LIN {X 0,Y 573.635,Z 572.354,A -85,B 0,C 180,E1 -2236.63,E2 -2236.63} C_VEL
LIN {X 0,Y 573.477,Z 582.752,A -85,B 0,C 180,E1 -2237.616,E2 -2237.616} C_VEL
LIN {X 0,Y 573.285,Z 592.771,A -85,B 0,C 180,E1 -2238.734,E2 -2238.734} C_VEL
LIN {X 0,Y 573.242,Z 601.859,A -85,B 0,C 180,E1 -2239.939,E2 -2239.939} C_VEL
LIN {X 0,Y 573.133,Z 609.735,A -85,B 0,C 180,E1 -2241.183,E2 -2241.183} C_VEL
LIN {X 0,Y 573.074,Z 617.09,A -85,B 0,C 180,E1 -2242.602,E2 -2242.602} C_VEL
LIN {X 0,Y 573.04,Z 622.924,A -85,B 0,C 180,E1 -2244.016,E2 -2244.016} C_VEL
LIN {X 0,Y 572.951,Z 626.386,A -85,B 0,C 180,E1 -2245.074,E2 -2245.074} C_VEL
LIN {X 0,Y 573.004,Z 629.889,A -85,B 0,C 180,E1 -2246.484,E2 -2246.484} C_VEL
LIN {X 0,Y 572.937,Z 632.192,A -85,B 0,C 180,E1 -2247.891,E2 -2247.891} C_VEL
LIN {X 0,Y 572.938,Z 633.349,A -85,B 0,C 180,E1 -2249.297,E2 -2249.297} C_VEL
LIN {X 0,Y 572.938,Z 633.349,A -85,B 0,C 180,E1 -2250.703,E2 -2250.703} C_VEL
LIN {X 0,Y 572.937,Z 632.191,A -85,B 0,C 180,E1 -2252.109,E2 -2252.109} C_VEL
LIN {X 0,Y 573.004,Z 629.887,A -85,B 0,C 180,E1 -2253.516,E2 -2253.516} C_VEL
LIN {X 0,Y 572.951,Z 626.386,A -85,B 0,C 180,E1 -2254.926,E2 -2254.926} C_VEL
LIN {X 0,Y 573.012,Z 621.609,A -85,B 0,C 180,E1 -2256.337,E2 -2256.337} C_VEL
LIN {X 0,Y 573.093,Z 615.424,A -85,B 0,C 180,E1 -2257.752,E2 -2257.752} C_VEL
LIN {X 0,Y 573.136,Z 607.65,A -85,B 0,C 180,E1 -2259.172,E2 -2259.172} C_VEL
LIN {X 0,Y 573.27,Z 599.371,A -85,B 0,C 180,E1 -2260.418,E2 -2260.418} C_VEL
LIN {X 0,Y 573.385,Z 589.394,A -85,B 0,C 180,E1 -2261.668,E2 -2261.668} C_VEL
LIN {X 0,Y 573.568,Z 579.192,A -85,B 0,C 180,E1 -2262.741,E2 -2262.741} C_VEL
LIN {X 0,Y 573.742,Z 567.024,A -85,B 0,C 180,E1 -2263.819,E2 -2263.819} C_VEL
LIN {X 0,Y 573.961,Z 553.91,A -85,B 0,C 180,E1 -2264.781,E2 -2264.781} C_VEL
LIN {X 0,Y 574.143,Z 539.88,A -85,B 0,C 180,E1 -2265.622,E2 -2265.622} C_VEL
LIN {X 0,Y 574.334,Z 525.81,A -85,B 0,C 180,E1 -2266.3,E2 -2266.3} C_VEL
LIN {X 0,Y 574.562,Z 511.319,A -85,B 0,C 180,E1 -2266.842,E2 -2266.842} C_VEL
LIN {X 0,Y 574.705,Z 496.022,A -85,B 0,C 180,E1 -2267.261,E2 -2267.261} C_VEL
LIN {X 0,Y 574.796,Z 480.66,A -85,B 0,C 180,E1 -2267.532,E2 -2267.532} C_VEL
LIN {X 0,Y 575.14,Z 327.837,A -85,B 0,C 180,E1 -2269.493,E2 -2269.493} C_VEL
LIN {X 0,Y 574.002,Z 321.813,A -85,B 0,C 180,E1 -2269.623,E2 -2269.623} C_VEL
LIN {X 0,Y 574.348,Z 296.397,A -85,B 0,C 180,E1 -2272.671,E2 -2272.671} C_VEL
LIN {X 0,Y 574.606,Z 274.457,A -85,B 0,C 180,E1 -2275.345,E2 -2275.345} C_VEL
LIN {X 0,Y 574.309,Z 271.29,A -85,B 0,C 180,E1 -2275.748,E2 -2275.748} C_VEL
LIN {X 0,Y 573.237,Z 266.71,A -85,B 0,C 180,E1 -2276.376,E2 -2276.376} C_VEL
LIN {X 0,Y 573.255,Z 266.699,A -85,B 0,C 180,E1 -2279.365,E2 -2279.365} C_VEL
LIN {X 0,Y 573.242,Z 266.707,A -85,B 0,C 180,E1 -2282.227,E2 -2282.227} C_VEL
LIN {X 0,Y 573.219,Z 266.703,A -85,B 0,C 180,E1 -2284.769,E2 -2284.769} C_VEL
LIN {X 0,Y 573.216,Z 266.708,A -85,B 0,C 180,E1 -2287.808,E2 -2287.808} C_VEL
LIN {X 0,Y 573.238,Z 266.703,A -85,B 0,C 180,E1 -2290.524,E2 -2290.524} C_VEL
LIN {X 0,Y 573.19,Z 266.707,A -85,B 0,C 180,E1 -2293.362,E2 -2293.362} C_VEL
LIN {X 0,Y 573.2,Z 266.709,A -85,B 0,C 180,E1 -2296.334,E2 -2296.334} C_VEL
LIN {X 0,Y 573.198,Z 266.706,A -85,B 0,C 180,E1 -2298.54,E2 -2298.54} C_VEL
LIN {X 0,Y 573.221,Z 266.703,A -85,B 0,C 180,E1 -2301.297,E2 -2301.297} C_VEL
LIN {X 0,Y 573.173,Z 266.715,A -85,B 0,C 180,E1 -2304.022,E2 -2304.022} C_VEL
LIN {X 0,Y 573.218,Z 266.702,A -85,B 0,C 180,E1 -2306.514,E2 -2306.514} C_VEL
LIN {X 0,Y 573.208,Z 266.704,A -85,B 0,C 180,E1 -2309.119,E2 -2309.119} C_VEL
LIN {X 0,Y 573.207,Z 266.709,A -85,B 0,C 180,E1 -2311.977,E2 -2311.977} C_VEL
LIN {X 0,Y 573.192,Z 266.705,A -85,B 0,C 180,E1 -2314.587,E2 -2314.587} C_VEL
LIN {X 0,Y 573.222,Z 266.702,A -85,B 0,C 180,E1 -2316.9,E2 -2316.9} C_VEL
LIN {X 0,Y 573.233,Z 266.703,A -85,B 0,C 180,E1 -2319.173,E2 -2319.173} C_VEL
LIN {X 0,Y 573.186,Z 266.709,A -85,B 0,C 180,E1 -2321.41,E2 -2321.41} C_VEL
LIN {X 0,Y 573.2,Z 266.705,A -85,B 0,C 180,E1 -2324.351,E2 -2324.351} C_VEL
LIN {X 0,Y 573.187,Z 266.705,A -85,B 0,C 180,E1 -2326.528,E2 -2326.528} C_VEL
LIN {X 0,Y 573.212,Z 266.706,A -85,B 0,C 180,E1 -2329.402,E2 -2329.402} C_VEL
LIN {X 0,Y 573.196,Z 266.705,A -85,B 0,C 180,E1 -2332.249,E2 -2332.249} C_VEL
LIN {X 0,Y 573.246,Z 266.697,A -85,B 0,C 180,E1 -2334.371,E2 -2334.371} C_VEL
LIN {X 0,Y 573.283,Z 266.7,A -85,B 0,C 180,E1 -2337.189,E2 -2337.189} C_VEL
LIN {X 0,Y 573.285,Z 266.695,A -85,B 0,C 180,E1 -2340,E2 -2340} C_VEL
LIN {X 0,Y 573.272,Z 266.697,A -85,B 0,C 180,E1 -2342.811,E2 -2342.811} C_VEL
LIN {X 0,Y 573.27,Z 266.7,A -85,B 0,C 180,E1 -2345.628,E2 -2345.628} C_VEL
LIN {X 0,Y 573.251,Z 266.701,A -85,B 0,C 180,E1 -2347.751,E2 -2347.751} C_VEL
LIN {X 0,Y 573.226,Z 266.702,A -85,B 0,C 180,E1 -2350.597,E2 -2350.597} C_VEL
LIN {X 0,Y 573.21,Z 266.706,A -85,B 0,C 180,E1 -2352.75,E2 -2352.75} C_VEL
LIN {X 0,Y 573.207,Z 266.709,A -85,B 0,C 180,E1 -2354.921,E2 -2354.921} C_VEL
LIN {X 0,Y 573.22,Z 266.702,A -85,B 0,C 180,E1 -2357.849,E2 -2357.849} C_VEL
LIN {X 0,Y 573.221,Z 266.698,A -85,B 0,C 180,E1 -2360.078,E2 -2360.078} C_VEL
LIN {X 0,Y 573.208,Z 266.702,A -85,B 0,C 180,E1 -2362.339,E2 -2362.339} C_VEL
LIN {X 0,Y 573.2,Z 266.705,A -85,B 0,C 180,E1 -2364.352,E2 -2364.352} C_VEL
LIN {X 0,Y 572.567,Z 266.791,A -85,B 0,C 180,E1 -2364.938,E2 -2364.938} C_VEL
LIN {X 0,Y 569.747,Z 267.143,A -85,B 0,C 180,E1 -2365.89,E2 -2365.89} C_VEL
LIN {X 0,Y 567.336,Z 267.442,A -85,B 0,C 180,E1 -2366.656,E2 -2366.656} C_VEL
LIN {X 0,Y 566.283,Z 267.569,A -85,B 0,C 180,E1 -2367.247,E2 -2367.247} C_VEL
LIN {X 0,Y 566.19,Z 267.578,A -85,B 0,C 180,E1 -2367.447,E2 -2367.447} C_VEL
LIN {X 0,Y 566.185,Z 267.578,A -85,B 0,C 180,E1 -2369.77,E2 -2369.77} C_VEL
LIN {X 0,Y 566.191,Z 267.579,A -85,B 0,C 180,E1 -2372.43,E2 -2372.43} C_VEL
LIN {X 0,Y 566.173,Z 267.588,A -85,B 0,C 180,E1 -2374.991,E2 -2374.991} C_VEL
LIN {X 0,Y 566.186,Z 267.579,A -85,B 0,C 180,E1 -2377.462,E2 -2377.462} C_VEL
LIN {X 0,Y 566.198,Z 267.577,A -85,B 0,C 180,E1 -2380.2,E2 -2380.2} C_VEL
LIN {X 0,Y 566.193,Z 267.583,A -85,B 0,C 180,E1 -2383.055,E2 -2383.055} C_VEL
LIN {X 0,Y 566.187,Z 267.579,A -85,B 0,C 180,E1 -2386.05,E2 -2386.05} C_VEL
LIN {X 0,Y 566.197,Z 267.58,A -85,B 0,C 180,E1 -2389.216,E2 -2389.216} C_VEL
LIN {X 0,Y 566.176,Z 267.579,A -85,B 0,C 180,E1 -2391.637,E2 -2391.637} C_VEL
LIN {X 0,Y 566.169,Z 267.585,A -85,B 0,C 180,E1 -2394.31,E2 -2394.31} C_VEL
LIN {X 0,Y 566.2,Z 267.583,A -85,B 0,C 180,E1 -2396.898,E2 -2396.898} C_VEL
LIN {X 0,Y 566.175,Z 267.581,A -85,B 0,C 180,E1 -2399.408,E2 -2399.408} C_VEL
LIN {X 0,Y 566.21,Z 267.577,A -85,B 0,C 180,E1 -2401.858,E2 -2401.858} C_VEL
LIN {X 0,Y 566.209,Z 267.582,A -85,B 0,C 180,E1 -2404.252,E2 -2404.252} C_VEL
LIN {X 0,Y 566.227,Z 267.735,A -85,B 0,C 180,E1 -2406.574,E2 -2406.574} C_VEL
LIN {X 0,Y 567.168,Z 273.21,A -85,B 0,C 180,E1 -2407.411,E2 -2407.411} C_VEL
LIN {X 0,Y 566.915,Z 292.519,A -85,B 0,C 180,E1 -2410.134,E2 -2410.134} C_VEL
LIN {X 0,Y 566.916,Z 292.904,A -85,B 0,C 180,E1 -2410.188,E2 -2410.188} C_VEL
LIN {X 0,Y 568.47,Z 301.087,A -85,B 0,C 180,E1 -2410.357,E2 -2410.357} C_VEL
LIN {X 0,Y 567.974,Z 458.169,A -85,B 0,C 180,E1 -2412.413,E2 -2412.413} C_VEL
LIN {X 0,Y 567.827,Z 473.784,A -85,B 0,C 180,E1 -2412.767,E2 -2412.767} C_VEL
LIN {X 0,Y 567.607,Z 489.09,A -85,B 0,C 180,E1 -2413.27,E2 -2413.27} C_VEL
LIN {X 0,Y 567.399,Z 503.742,A -85,B 0,C 180,E1 -2413.911,E2 -2413.911} C_VEL
LIN {X 0,Y 567.146,Z 517.054,A -85,B 0,C 180,E1 -2414.641,E2 -2414.641} C_VEL
LIN {X 0,Y 566.917,Z 529.984,A -85,B 0,C 180,E1 -2415.508,E2 -2415.508} C_VEL
LIN {X 0,Y 566.653,Z 542.893,A -85,B 0,C 180,E1 -2416.553,E2 -2416.553} C_VEL
LIN {X 0,Y 566.479,Z 554.088,A -85,B 0,C 180,E1 -2417.643,E2 -2417.643} C_VEL
LIN {X 0,Y 566.263,Z 564.18,A -85,B 0,C 180,E1 -2418.81,E2 -2418.81} C_VEL
LIN {X 0,Y 566.133,Z 574.006,A -85,B 0,C 180,E1 -2420.172,E2 -2420.172} C_VEL
LIN {X 0,Y 566.064,Z 581.496,A -85,B 0,C 180,E1 -2421.432,E2 -2421.432} C_VEL
LIN {X 0,Y 565.975,Z 588.5,A -85,B 0,C 180,E1 -2422.867,E2 -2422.867} C_VEL
LIN {X 0,Y 565.981,Z 594.009,A -85,B 0,C 180,E1 -2424.299,E2 -2424.299} C_VEL
LIN {X 0,Y 565.914,Z 598.178,A -85,B 0,C 180,E1 -2425.727,E2 -2425.727} C_VEL
LIN {X 0,Y 565.872,Z 601.113,A -85,B 0,C 180,E1 -2427.153,E2 -2427.153} C_VEL
LIN {X 0,Y 565.842,Z 602.879,A -85,B 0,C 180,E1 -2428.577,E2 -2428.577} C_VEL
LIN {X 0,Y 565.837,Z 603.496,A -85,B 0,C 180,E1 -2430,E2 -2430} C_VEL
LIN {X 0,Y 565.844,Z 602.941,A -85,B 0,C 180,E1 -2431.423,E2 -2431.423} C_VEL
LIN {X 0,Y 565.874,Z 601.258,A -85,B 0,C 180,E1 -2432.847,E2 -2432.847} C_VEL
LIN {X 0,Y 565.914,Z 598.404,A -85,B 0,C 180,E1 -2434.273,E2 -2434.273} C_VEL
LIN {X 0,Y 565.975,Z 594.318,A -85,B 0,C 180,E1 -2435.701,E2 -2435.701} C_VEL
LIN {X 0,Y 565.975,Z 588.904,A -85,B 0,C 180,E1 -2437.133,E2 -2437.133} C_VEL
LIN {X 0,Y 566.06,Z 582.004,A -85,B 0,C 180,E1 -2438.568,E2 -2438.568} C_VEL
LIN {X 0,Y 566.177,Z 573.396,A -85,B 0,C 180,E1 -2440.008,E2 -2440.008} C_VEL
LIN {X 0,Y 566.25,Z 564.953,A -85,B 0,C 180,E1 -2441.183,E2 -2441.183} C_VEL
LIN {X 0,Y 566.436,Z 554.917,A -85,B 0,C 180,E1 -2442.358,E2 -2442.358} C_VEL
LIN {X 0,Y 566.668,Z 542.874,A -85,B 0,C 180,E1 -2443.538,E2 -2443.538} C_VEL
LIN {X 0,Y 566.877,Z 531.252,A -85,B 0,C 180,E1 -2444.488,E2 -2444.488} C_VEL
LIN {X 0,Y 567.09,Z 518.478,A -85,B 0,C 180,E1 -2445.361,E2 -2445.361} C_VEL
LIN {X 0,Y 567.377,Z 505.469,A -85,B 0,C 180,E1 -2446.09,E2 -2446.09} C_VEL
LIN {X 0,Y 567.555,Z 491.278,A -85,B 0,C 180,E1 -2446.732,E2 -2446.732} C_VEL
LIN {X 0,Y 567.793,Z 476.732,A -85,B 0,C 180,E1 -2447.235,E2 -2447.235} C_VEL
LIN {X 0,Y 567.922,Z 461.44,A -85,B 0,C 180,E1 -2447.613,E2 -2447.613} C_VEL
LIN {X 0,Y 568.073,Z 439.94,A -85,B 0,C 180,E1 -2447.931,E2 -2447.931} C_VEL
LIN {X 0,Y 568.46,Z 300.582,A -85,B 0,C 180,E1 -2449.74,E2 -2449.74} C_VEL
LIN {X 0,Y 566.883,Z 292.906,A -85,B 0,C 180,E1 -2449.903,E2 -2449.903} C_VEL
LIN {X 0,Y 567.205,Z 275.173,A -85,B 0,C 180,E1 -2452.396,E2 -2452.396} C_VEL
LIN {X 0,Y 566.947,Z 271.258,A -85,B 0,C 180,E1 -2452.973,E2 -2452.973} C_VEL
LIN {X 0,Y 566.211,Z 267.584,A -85,B 0,C 180,E1 -2453.548,E2 -2453.548} C_VEL
LIN {X 0,Y 566.213,Z 267.583,A -85,B 0,C 180,E1 -2455.748,E2 -2455.748} C_VEL
LIN {X 0,Y 566.201,Z 267.579,A -85,B 0,C 180,E1 -2458.201,E2 -2458.201} C_VEL
LIN {X 0,Y 566.191,Z 267.582,A -85,B 0,C 180,E1 -2461.076,E2 -2461.076} C_VEL
LIN {X 0,Y 566.209,Z 267.581,A -85,B 0,C 180,E1 -2463.733,E2 -2463.733} C_VEL
LIN {X 0,Y 566.204,Z 267.577,A -85,B 0,C 180,E1 -2466.568,E2 -2466.568} C_VEL
LIN {X 0,Y 566.215,Z 267.578,A -85,B 0,C 180,E1 -2469.686,E2 -2469.686} C_VEL
LIN {X 0,Y 566.195,Z 267.581,A -85,B 0,C 180,E1 -2472.916,E2 -2472.916} C_VEL
LIN {X 0,Y 566.186,Z 267.579,A -85,B 0,C 180,E1 -2476.048,E2 -2476.048} C_VEL
LIN {X 0,Y 566.195,Z 267.584,A -85,B 0,C 180,E1 -2479.214,E2 -2479.214} C_VEL
LIN {X 0,Y 566.173,Z 267.582,A -85,B 0,C 180,E1 -2481.636,E2 -2481.636} C_VEL
LIN {X 0,Y 566.155,Z 267.58,A -85,B 0,C 180,E1 -2484.307,E2 -2484.307} C_VEL
LIN {X 0,Y 566.193,Z 267.583,A -85,B 0,C 180,E1 -2486.896,E2 -2486.896} C_VEL
LIN {X 0,Y 566.167,Z 267.582,A -85,B 0,C 180,E1 -2489.406,E2 -2489.406} C_VEL
LIN {X 0,Y 566.201,Z 267.576,A -85,B 0,C 180,E1 -2491.857,E2 -2491.857} C_VEL
LIN {X 0,Y 566.193,Z 267.577,A -85,B 0,C 180,E1 -2494.25,E2 -2494.25} C_VEL
LIN {X 0,Y 566.159,Z 267.584,A -85,B 0,C 180,E1 -2497.367,E2 -2497.367} C_VEL
LIN {X 0,Y 566.191,Z 267.578,A -85,B 0,C 180,E1 -2499.662,E2 -2499.662} C_VEL
LIN {X 0,Y 566.183,Z 267.583,A -85,B 0,C 180,E1 -2502.668,E2 -2502.668} C_VEL
LIN {X 0,Y 566.2,Z 267.576,A -85,B 0,C 180,E1 -2505.626,E2 -2505.626} C_VEL
LIN {X 0,Y 566.219,Z 267.581,A -85,B 0,C 180,E1 -2508.676,E2 -2508.676} C_VEL
LIN {X 0,Y 566.178,Z 267.579,A -85,B 0,C 180,E1 -2511.433,E2 -2511.433} C_VEL
LIN {X 0,Y 566.237,Z 267.575,A -85,B 0,C 180,E1 -2514.301,E2 -2514.301} C_VEL
LIN {X 0,Y 566.248,Z 267.571,A -85,B 0,C 180,E1 -2517.866,E2 -2517.866} C_VEL
LIN {X 0,Y 566.291,Z 267.574,A -85,B 0,C 180,E1 -2520.711,E2 -2520.711} C_VEL
LIN {X 0,Y 566.25,Z 267.576,A -85,B 0,C 180,E1 -2522.846,E2 -2522.846} C_VEL
LIN {X 0,Y 566.217,Z 267.574,A -85,B 0,C 180,E1 -2525.699,E2 -2525.699} C_VEL
LIN {X 0,Y 566.168,Z 267.581,A -85,B 0,C 180,E1 -2527.848,E2 -2527.848} C_VEL
LIN {X 0,Y 566.205,Z 267.582,A -85,B 0,C 180,E1 -2530.73,E2 -2530.73} C_VEL
LIN {X 0,Y 566.163,Z 267.58,A -85,B 0,C 180,E1 -2533.642,E2 -2533.642} C_VEL
LIN {X 0,Y 566.168,Z 267.582,A -85,B 0,C 180,E1 -2535.848,E2 -2535.848} C_VEL
LIN {X 0,Y 566.173,Z 267.583,A -85,B 0,C 180,E1 -2538.829,E2 -2538.829} C_VEL
LIN {X 0,Y 566.194,Z 267.577,A -85,B 0,C 180,E1 -2541.42,E2 -2541.42} C_VEL
LIN {X 0,Y 566.155,Z 267.59,A -85,B 0,C 180,E1 -2544.183,E2 -2544.183} C_VEL
LIN {X 0,Y 566.155,Z 267.586,A -85,B 0,C 180,E1 -2546.652,E2 -2546.652} C_VEL
LIN {X 0,Y 566.157,Z 267.583,A -85,B 0,C 180,E1 -2548.955,E2 -2548.955} C_VEL
LIN {X 0,Y 566.176,Z 267.58,A -85,B 0,C 180,E1 -2551.423,E2 -2551.423} C_VEL
LIN {X 0,Y 566.181,Z 267.584,A -85,B 0,C 180,E1 -2553.958,E2 -2553.958} C_VEL
LIN {X 0,Y 566.133,Z 267.588,A -85,B 0,C 180,E1 -2556.575,E2 -2556.575} C_VEL
LIN {X 0,Y 566.195,Z 267.576,A -85,B 0,C 180,E1 -2559.275,E2 -2559.275} C_VEL
LIN {X 0,Y 566.172,Z 267.588,A -85,B 0,C 180,E1 -2562.091,E2 -2562.091} C_VEL
LIN {X 0,Y 566.154,Z 267.582,A -85,B 0,C 180,E1 -2565.038,E2 -2565.038} C_VEL
LIN {X 0,Y 566.161,Z 267.59,A -85,B 0,C 180,E1 -2567.909,E2 -2567.909} C_VEL
LIN {X 0,Y 566.202,Z 267.577,A -85,B 0,C 180,E1 -2570.727,E2 -2570.727} C_VEL
LIN {X 0,Y 566.171,Z 267.583,A -85,B 0,C 180,E1 -2573.429,E2 -2573.429} C_VEL
LIN {X 0,Y 566.206,Z 267.58,A -85,B 0,C 180,E1 -2576.267,E2 -2576.267} C_VEL
LIN {X 0,Y 566.183,Z 267.579,A -85,B 0,C 180,E1 -2578.925,E2 -2578.925} C_VEL
LIN {X 0,Y 566.183,Z 267.588,A -85,B 0,C 180,E1 -2581.857,E2 -2581.857} C_VEL
LIN {X 0,Y 566.163,Z 267.651,A -85,B 0,C 180,E1 -2583.424,E2 -2583.424} C_VEL
LIN {X 0,Y 567.691,Z 274.277,A -85,B 0,C 180,E1 -2584.324,E2 -2584.324} C_VEL
LIN {X 0,Y 567.568,Z 291.067,A -85,B 0,C 180,E1 -2586.393,E2 -2586.393} C_VEL
LIN {X 0,Y 567.282,Z 312.003,A -85,B 0,C 180,E1 -2588.945,E2 -2588.945} C_VEL
LIN {X 0,Y 567.116,Z 321.949,A -85,B 0,C 180,E1 -2590.143,E2 -2590.143} C_VEL
LIN {X 0,Y 568.507,Z 330.374,A -85,B 0,C 180,E1 -2590.304,E2 -2590.304} C_VEL
LIN {X 0,Y 567.994,Z 488.201,A -85,B 0,C 180,E1 -2592.369,E2 -2592.369} C_VEL
LIN {X 0,Y 567.834,Z 503.721,A -85,B 0,C 180,E1 -2592.72,E2 -2592.72} C_VEL
LIN {X 0,Y 567.61,Z 519.05,A -85,B 0,C 180,E1 -2593.223,E2 -2593.223} C_VEL
LIN {X 0,Y 567.444,Z 532.784,A -85,B 0,C 180,E1 -2593.82,E2 -2593.82} C_VEL
LIN {X 0,Y 567.151,Z 546.255,A -85,B 0,C 180,E1 -2594.549,E2 -2594.549} C_VEL
LIN {X 0,Y 566.931,Z 558.527,A -85,B 0,C 180,E1 -2595.359,E2 -2595.359} C_VEL
LIN {X 0,Y 566.671,Z 571.296,A -85,B 0,C 180,E1 -2596.371,E2 -2596.371} C_VEL
LIN {X 0,Y 566.491,Z 582.753,A -85,B 0,C 180,E1 -2597.461,E2 -2597.461} C_VEL
LIN {X 0,Y 566.268,Z 593.314,A -85,B 0,C 180,E1 -2598.659,E2 -2598.659} C_VEL
LIN {X 0,Y 566.208,Z 601.858,A -85,B 0,C 180,E1 -2599.812,E2 -2599.812} C_VEL
LIN {X 0,Y 566.057,Z 609.736,A -85,B 0,C 180,E1 -2601.072,E2 -2601.072} C_VEL
LIN {X 0,Y 565.997,Z 617.091,A -85,B 0,C 180,E1 -2602.509,E2 -2602.509} C_VEL
LIN {X 0,Y 565.956,Z 622.923,A -85,B 0,C 180,E1 -2603.941,E2 -2603.941} C_VEL
LIN {X 0,Y 565.866,Z 626.386,A -85,B 0,C 180,E1 -2605.013,E2 -2605.013} C_VEL
LIN {X 0,Y 565.909,Z 629.89,A -85,B 0,C 180,E1 -2606.44,E2 -2606.44} C_VEL
LIN {X 0,Y 565.838,Z 632.192,A -85,B 0,C 180,E1 -2607.865,E2 -2607.865} C_VEL
LIN {X 0,Y 565.838,Z 633.349,A -85,B 0,C 180,E1 -2609.288,E2 -2609.288} C_VEL
LIN {X 0,Y 565.838,Z 633.348,A -85,B 0,C 180,E1 -2610.712,E2 -2610.712} C_VEL
LIN {X 0,Y 565.838,Z 632.19,A -85,B 0,C 180,E1 -2612.135,E2 -2612.135} C_VEL
LIN {X 0,Y 565.909,Z 629.887,A -85,B 0,C 180,E1 -2613.56,E2 -2613.56} C_VEL
LIN {X 0,Y 565.866,Z 626.386,A -85,B 0,C 180,E1 -2614.987,E2 -2614.987} C_VEL
LIN {X 0,Y 565.956,Z 622.925,A -85,B 0,C 180,E1 -2616.059,E2 -2616.059} C_VEL
LIN {X 0,Y 565.997,Z 617.089,A -85,B 0,C 180,E1 -2617.491,E2 -2617.491} C_VEL
LIN {X 0,Y 566.057,Z 609.732,A -85,B 0,C 180,E1 -2618.928,E2 -2618.928} C_VEL
LIN {X 0,Y 566.208,Z 601.858,A -85,B 0,C 180,E1 -2620.188,E2 -2620.188} C_VEL
LIN {X 0,Y 566.308,Z 592.393,A -85,B 0,C 180,E1 -2621.453,E2 -2621.453} C_VEL
LIN {X 0,Y 566.491,Z 582.752,A -85,B 0,C 180,E1 -2622.539,E2 -2622.539} C_VEL
LIN {X 0,Y 566.672,Z 571.299,A -85,B 0,C 180,E1 -2623.629,E2 -2623.629} C_VEL
LIN {X 0,Y 566.948,Z 558.683,A -85,B 0,C 180,E1 -2624.63,E2 -2624.63} C_VEL
LIN {X 0,Y 567.151,Z 546.253,A -85,B 0,C 180,E1 -2625.451,E2 -2625.451} C_VEL
LIN {X 0,Y 567.461,Z 532.778,A -85,B 0,C 180,E1 -2626.18,E2 -2626.18} C_VEL
LIN {X 0,Y 567.639,Z 519.058,A -85,B 0,C 180,E1 -2626.776,E2 -2626.776} C_VEL
LIN {X 0,Y 567.847,Z 503.735,A -85,B 0,C 180,E1 -2627.279,E2 -2627.279} C_VEL
LIN {X 0,Y 567.98,Z 488.315,A -85,B 0,C 180,E1 -2627.63,E2 -2627.63} C_VEL
LIN {X 0,Y 568.493,Z 329.51,A -85,B 0,C 180,E1 -2629.708,E2 -2629.708} C_VEL
LIN {X 0,Y 567.135,Z 321.838,A -85,B 0,C 180,E1 -2629.867,E2 -2629.867} C_VEL
LIN {X 0,Y 567.548,Z 294.798,A -85,B 0,C 180,E1 -2633.151,E2 -2633.151} C_VEL
LIN {X 0,Y 567.795,Z 276.046,A -85,B 0,C 180,E1 -2635.452,E2 -2635.452} C_VEL
LIN {X 0,Y 567.025,Z 271.103,A -85,B 0,C 180,E1 -2636.103,E2 -2636.103} C_VEL
LIN {X 0,Y 566.15,Z 267.591,A -85,B 0,C 180,E1 -2636.598,E2 -2636.598} C_VEL
LIN {X 0,Y 566.178,Z 267.581,A -85,B 0,C 180,E1 -2638.953,E2 -2638.953} C_VEL
LIN {X 0,Y 566.185,Z 267.579,A -85,B 0,C 180,E1 -2641.421,E2 -2641.421} C_VEL
LIN {X 0,Y 566.202,Z 267.584,A -85,B 0,C 180,E1 -2643.955,E2 -2643.955} C_VEL
LIN {X 0,Y 566.171,Z 267.583,A -85,B 0,C 180,E1 -2646.571,E2 -2646.571} C_VEL
LIN {X 0,Y 566.204,Z 267.581,A -85,B 0,C 180,E1 -2649.684,E2 -2649.684} C_VEL
LIN {X 0,Y 566.174,Z 267.58,A -85,B 0,C 180,E1 -2652.914,E2 -2652.914} C_VEL
LIN {X 0,Y 566.15,Z 267.592,A -85,B 0,C 180,E1 -2656.052,E2 -2656.052} C_VEL
LIN {X 0,Y 566.149,Z 267.583,A -85,B 0,C 180,E1 -2658.858,E2 -2658.858} C_VEL
LIN {X 0,Y 566.191,Z 267.581,A -85,B 0,C 180,E1 -2661.442,E2 -2661.442} C_VEL
LIN {X 0,Y 566.128,Z 267.588,A -85,B 0,C 180,E1 -2664.305,E2 -2664.305} C_VEL
LIN {X 0,Y 566.187,Z 267.577,A -85,B 0,C 180,E1 -2666.896,E2 -2666.896} C_VEL
LIN {X 0,Y 566.157,Z 267.585,A -85,B 0,C 180,E1 -2669.406,E2 -2669.406} C_VEL
LIN {X 0,Y 566.174,Z 267.587,A -85,B 0,C 180,E1 -2671.855,E2 -2671.855} C_VEL
LIN {X 0,Y 566.161,Z 267.583,A -85,B 0,C 180,E1 -2674.249,E2 -2674.249} C_VEL
LIN {X 0,Y 566.152,Z 267.582,A -85,B 0,C 180,E1 -2676.72,E2 -2676.72} C_VEL
LIN {X 0,Y 566.187,Z 267.585,A -85,B 0,C 180,E1 -2679.662,E2 -2679.662} C_VEL
LIN {X 0,Y 566.154,Z 267.586,A -85,B 0,C 180,E1 -2681.92,E2 -2681.92} C_VEL
LIN {X 0,Y 566.173,Z 267.581,A -85,B 0,C 180,E1 -2684.89,E2 -2684.89} C_VEL
LIN {X 0,Y 566.162,Z 267.581,A -85,B 0,C 180,E1 -2687.817,E2 -2687.817} C_VEL
LIN {X 0,Y 566.125,Z 267.587,A -85,B 0,C 180,E1 -2689.991,E2 -2689.991} C_VEL
LIN {X 0,Y 566.218,Z 267.576,A -85,B 0,C 180,E1 -2692.87,E2 -2692.87} C_VEL
LIN {X 0,Y 566.258,Z 267.571,A -85,B 0,C 180,E1 -2695.016,E2 -2695.016} C_VEL
LIN {X 0,Y 566.249,Z 267.572,A -85,B 0,C 180,E1 -2697.866,E2 -2697.866} C_VEL
LIN {X 0,Y 566.256,Z 267.571,A -85,B 0,C 180,E1 -2700,E2 -2700} C_VEL
LIN {X 0,Y 566.241,Z 267.573,A -85,B 0,C 180,E1 -2702.846,E2 -2702.846} C_VEL
LIN {X 0,Y 566.235,Z 267.575,A -85,B 0,C 180,E1 -2705.699,E2 -2705.699} C_VEL
LIN {X 0,Y 566.177,Z 267.58,A -85,B 0,C 180,E1 -2708.567,E2 -2708.567} C_VEL
LIN {X 0,Y 566.227,Z 267.579,A -85,B 0,C 180,E1 -2711.455,E2 -2711.455} C_VEL
LIN {X 0,Y 566.191,Z 267.578,A -85,B 0,C 180,E1 -2714.495,E2 -2714.495} C_VEL
LIN {X 0,Y 566.178,Z 267.585,A -85,B 0,C 180,E1 -2717.332,E2 -2717.332} C_VEL
LIN {X 0,Y 566.186,Z 267.577,A -85,B 0,C 180,E1 -2719.582,E2 -2719.582} C_VEL
LIN {X 0,Y 566.173,Z 267.578,A -85,B 0,C 180,E1 -2721.863,E2 -2721.863} C_VEL
LIN {X 0,Y 566.171,Z 267.589,A -85,B 0,C 180,E1 -2725.023,E2 -2725.023} C_VEL
LIN {X 0,Y 566.19,Z 267.578,A -85,B 0,C 180,E1 -2727.447,E2 -2727.447} C_VEL
LIN {X 0,Y 565.5,Z 267.663,A -85,B 0,C 180,E1 -2728.041,E2 -2728.041} C_VEL
LIN {X 0,Y 562.634,Z 268.028,A -85,B 0,C 180,E1 -2729.004,E2 -2729.004} C_VEL
LIN {X 0,Y 560.231,Z 268.323,A -85,B 0,C 180,E1 -2729.78,E2 -2729.78} C_VEL
LIN {X 0,Y 559.206,Z 268.449,A -85,B 0,C 180,E1 -2730.379,E2 -2730.379} C_VEL
LIN {X 0,Y 559.126,Z 268.46,A -85,B 0,C 180,E1 -2730.582,E2 -2730.582} C_VEL
LIN {X 0,Y 559.141,Z 268.461,A -85,B 0,C 180,E1 -2732.716,E2 -2732.716} C_VEL
LIN {X 0,Y 559.119,Z 268.462,A -85,B 0,C 180,E1 -2735.325,E2 -2735.325} C_VEL
LIN {X 0,Y 559.121,Z 268.458,A -85,B 0,C 180,E1 -2738.019,E2 -2738.019} C_VEL
LIN {X 0,Y 559.147,Z 268.464,A -85,B 0,C 180,E1 -2740.813,E2 -2740.813} C_VEL
LIN {X 0,Y 559.13,Z 268.457,A -85,B 0,C 180,E1 -2743.735,E2 -2743.735} C_VEL
LIN {X 0,Y 559.138,Z 268.465,A -85,B 0,C 180,E1 -2746.805,E2 -2746.805} C_VEL
LIN {X 0,Y 559.149,Z 268.458,A -85,B 0,C 180,E1 -2749.188,E2 -2749.188} C_VEL
LIN {X 0,Y 559.125,Z 268.458,A -85,B 0,C 180,E1 -2751.983,E2 -2751.983} C_VEL
LIN {X 0,Y 559.137,Z 268.465,A -85,B 0,C 180,E1 -2754.787,E2 -2754.787} C_VEL
LIN {X 0,Y 559.151,Z 268.456,A -85,B 0,C 180,E1 -2757.366,E2 -2757.366} C_VEL
LIN {X 0,Y 559.142,Z 268.46,A -85,B 0,C 180,E1 -2760.144,E2 -2760.144} C_VEL
LIN {X 0,Y 559.169,Z 268.454,A -85,B 0,C 180,E1 -2763.173,E2 -2763.173} C_VEL
LIN {X 0,Y 559.154,Z 268.458,A -85,B 0,C 180,E1 -2765.496,E2 -2765.496} C_VEL
LIN {X 0,Y 559.169,Z 268.524,A -85,B 0,C 180,E1 -2766.351,E2 -2766.351} C_VEL
LIN {X 0,Y 560.29,Z 274.712,A -85,B 0,C 180,E1 -2767.313,E2 -2767.313} C_VEL
LIN {X 0,Y 560.002,Z 292.91,A -85,B 0,C 180,E1 -2769.933,E2 -2769.933} C_VEL
LIN {X 0,Y 561.788,Z 302.213,A -85,B 0,C 180,E1 -2770.128,E2 -2770.128} C_VEL
LIN {X 0,Y 561.218,Z 458.437,A -85,B 0,C 180,E1 -2772.198,E2 -2772.198} C_VEL
LIN {X 0,Y 561.058,Z 473.804,A -85,B 0,C 180,E1 -2772.552,E2 -2772.552} C_VEL
LIN {X 0,Y 560.822,Z 489.103,A -85,B 0,C 180,E1 -2773.061,E2 -2773.061} C_VEL
LIN {X 0,Y 560.561,Z 503.751,A -85,B 0,C 180,E1 -2773.709,E2 -2773.709} C_VEL
LIN {X 0,Y 560.242,Z 517.065,A -85,B 0,C 180,E1 -2774.447,E2 -2774.447} C_VEL
LIN {X 0,Y 559.983,Z 530.396,A -85,B 0,C 180,E1 -2775.354,E2 -2775.354} C_VEL
LIN {X 0,Y 559.69,Z 542.9,A -85,B 0,C 180,E1 -2776.383,E2 -2776.383} C_VEL
LIN {X 0,Y 559.489,Z 554.094,A -85,B 0,C 180,E1 -2777.486,E2 -2777.486} C_VEL
LIN {X 0,Y 559.228,Z 564.79,A -85,B 0,C 180,E1 -2778.743,E2 -2778.743} C_VEL
LIN {X 0,Y 559.095,Z 574.009,A -85,B 0,C 180,E1 -2780.047,E2 -2780.047} C_VEL
LIN {X 0,Y 559.002,Z 581.498,A -85,B 0,C 180,E1 -2781.323,E2 -2781.323} C_VEL
LIN {X 0,Y 558.901,Z 588.502,A -85,B 0,C 180,E1 -2782.776,E2 -2782.776} C_VEL
LIN {X 0,Y 558.887,Z 594.011,A -85,B 0,C 180,E1 -2784.226,E2 -2784.226} C_VEL
LIN {X 0,Y 558.809,Z 598.179,A -85,B 0,C 180,E1 -2785.672,E2 -2785.672} C_VEL
LIN {X 0,Y 558.793,Z 601.113,A -85,B 0,C 180,E1 -2787.116,E2 -2787.116} C_VEL
LIN {X 0,Y 558.742,Z 602.879,A -85,B 0,C 180,E1 -2788.559,E2 -2788.559} C_VEL
LIN {X 0,Y 558.738,Z 603.496,A -85,B 0,C 180,E1 -2790,E2 -2790} C_VEL
LIN {X 0,Y 558.744,Z 602.94,A -85,B 0,C 180,E1 -2791.441,E2 -2791.441} C_VEL
LIN {X 0,Y 558.795,Z 601.256,A -85,B 0,C 180,E1 -2792.884,E2 -2792.884} C_VEL
LIN {X 0,Y 558.809,Z 598.403,A -85,B 0,C 180,E1 -2794.328,E2 -2794.328} C_VEL
LIN {X 0,Y 558.881,Z 594.317,A -85,B 0,C 180,E1 -2795.774,E2 -2795.774} C_VEL
LIN {X 0,Y 558.9,Z 588.901,A -85,B 0,C 180,E1 -2797.224,E2 -2797.224} C_VEL
LIN {X 0,Y 559,Z 582,A -85,B 0,C 180,E1 -2798.677,E2 -2798.677} C_VEL
LIN {X 0,Y 559.091,Z 574.573,A -85,B 0,C 180,E1 -2799.953,E2 -2799.953} C_VEL
LIN {X 0,Y 559.215,Z 565.512,A -85,B 0,C 180,E1 -2801.25,E2 -2801.25} C_VEL
LIN {X 0,Y 559.451,Z 554.912,A -85,B 0,C 180,E1 -2802.515,E2 -2802.515} C_VEL
LIN {X 0,Y 559.696,Z 542.868,A -85,B 0,C 180,E1 -2803.71,E2 -2803.71} C_VEL
LIN {X 0,Y 559.998,Z 530.177,A -85,B 0,C 180,E1 -2804.751,E2 -2804.751} C_VEL
LIN {X 0,Y 560.264,Z 517.013,A -85,B 0,C 180,E1 -2805.646,E2 -2805.646} C_VEL
LIN {X 0,Y 560.576,Z 503.689,A -85,B 0,C 180,E1 -2806.384,E2 -2806.384} C_VEL
LIN {X 0,Y 560.816,Z 489,A -85,B 0,C 180,E1 -2807.033,E2 -2807.033} C_VEL
LIN {X 0,Y 561.074,Z 473.522,A -85,B 0,C 180,E1 -2807.545,E2 -2807.545} C_VEL
LIN {X 0,Y 561.218,Z 457.604,A -85,B 0,C 180,E1 -2807.906,E2 -2807.906} C_VEL
LIN {X 0,Y 561.786,Z 301.668,A -85,B 0,C 180,E1 -2809.969,E2 -2809.969} C_VEL
LIN {X 0,Y 559.994,Z 292.791,A -85,B 0,C 180,E1 -2810.175,E2 -2810.175} C_VEL
LIN {X 0,Y 560.323,Z 275.357,A -85,B 0,C 180,E1 -2812.686,E2 -2812.686} C_VEL
LIN {X 0,Y 559.151,Z 268.464,A -85,B 0,C 180,E1 -2813.765,E2 -2813.765} C_VEL
LIN {X 0,Y 559.18,Z 268.455,A -85,B 0,C 180,E1 -2816.096,E2 -2816.096} C_VEL
LIN {X 0,Y 559.137,Z 268.458,A -85,B 0,C 180,E1 -2818.53,E2 -2818.53} C_VEL
LIN {X 0,Y 559.147,Z 268.463,A -85,B 0,C 180,E1 -2821.273,E2 -2821.273} C_VEL
LIN {X 0,Y 559.164,Z 268.456,A -85,B 0,C 180,E1 -2823.948,E2 -2823.948} C_VEL
LIN {X 0,Y 559.155,Z 268.456,A -85,B 0,C 180,E1 -2826.446,E2 -2826.446} C_VEL
LIN {X 0,Y 559.171,Z 268.456,A -85,B 0,C 180,E1 -2828.933,E2 -2828.933} C_VEL
LIN {X 0,Y 559.156,Z 268.458,A -85,B 0,C 180,E1 -2831.769,E2 -2831.769} C_VEL
LIN {X 0,Y 559.125,Z 268.46,A -85,B 0,C 180,E1 -2834.739,E2 -2834.739} C_VEL
LIN {X 0,Y 559.15,Z 268.462,A -85,B 0,C 180,E1 -2837.255,E2 -2837.255} C_VEL
LIN {X 0,Y 559.17,Z 268.452,A -85,B 0,C 180,E1 -2840.133,E2 -2840.133} C_VEL
LIN {X 0,Y 559.132,Z 268.461,A -85,B 0,C 180,E1 -2842.891,E2 -2842.891} C_VEL
LIN {X 0,Y 559.147,Z 268.455,A -85,B 0,C 180,E1 -2846.051,E2 -2846.051} C_VEL
LIN {X 0,Y 559.145,Z 268.46,A -85,B 0,C 180,E1 -2848.98,E2 -2848.98} C_VEL
LIN {X 0,Y 559.134,Z 268.458,A -85,B 0,C 180,E1 -2851.623,E2 -2851.623} C_VEL
LIN {X 0,Y 559.164,Z 268.452,A -85,B 0,C 180,E1 -2853.902,E2 -2853.902} C_VEL
LIN {X 0,Y 559.104,Z 268.468,A -85,B 0,C 180,E1 -2857.066,E2 -2857.066} C_VEL
LIN {X 0,Y 559.161,Z 268.456,A -85,B 0,C 180,E1 -2859.395,E2 -2859.395} C_VEL
LIN {X 0,Y 559.122,Z 268.458,A -85,B 0,C 180,E1 -2861.685,E2 -2861.685} C_VEL
LIN {X 0,Y 559.145,Z 268.455,A -85,B 0,C 180,E1 -2863.947,E2 -2863.947} C_VEL
LIN {X 0,Y 559.144,Z 268.456,A -85,B 0,C 180,E1 -2866.183,E2 -2866.183} C_VEL
LIN {X 0,Y 559.19,Z 268.455,A -85,B 0,C 180,E1 -2868.606,E2 -2868.606} C_VEL
LIN {X 0,Y 559.175,Z 268.451,A -85,B 0,C 180,E1 -2872.053,E2 -2872.053} C_VEL
LIN {X 0,Y 559.226,Z 268.449,A -85,B 0,C 180,E1 -2874.953,E2 -2874.953} C_VEL
LIN {X 0,Y 559.221,Z 268.446,A -85,B 0,C 180,E1 -2877.839,E2 -2877.839} C_VEL
LIN {X 0,Y 559.26,Z 268.449,A -85,B 0,C 180,E1 -2880.72,E2 -2880.72} C_VEL
LIN {X 0,Y 559.214,Z 268.452,A -85,B 0,C 180,E1 -2882.881,E2 -2882.881} C_VEL
LIN {X 0,Y 559.189,Z 268.449,A -85,B 0,C 180,E1 -2885.771,E2 -2885.771} C_VEL
LIN {X 0,Y 559.122,Z 268.46,A -85,B 0,C 180,E1 -2887.947,E2 -2887.947} C_VEL
LIN {X 0,Y 559.166,Z 268.457,A -85,B 0,C 180,E1 -2890.867,E2 -2890.867} C_VEL
LIN {X 0,Y 559.142,Z 268.455,A -85,B 0,C 180,E1 -2893.817,E2 -2893.817} C_VEL
LIN {X 0,Y 559.128,Z 268.461,A -85,B 0,C 180,E1 -2896.804,E2 -2896.804} C_VEL
LIN {X 0,Y 559.148,Z 268.457,A -85,B 0,C 180,E1 -2899.838,E2 -2899.838} C_VEL
LIN {X 0,Y 559.122,Z 268.464,A -85,B 0,C 180,E1 -2902.154,E2 -2902.154} C_VEL
LIN {X 0,Y 559.124,Z 268.457,A -85,B 0,C 180,E1 -2905.178,E2 -2905.178} C_VEL
LIN {X 0,Y 559.12,Z 268.466,A -85,B 0,C 180,E1 -2908.375,E2 -2908.375} C_VEL
LIN {X 0,Y 559.129,Z 268.457,A -85,B 0,C 180,E1 -2911.273,E2 -2911.273} C_VEL
LIN {X 0,Y 559.14,Z 268.46,A -85,B 0,C 180,E1 -2913.947,E2 -2913.947} C_VEL
LIN {X 0,Y 559.101,Z 268.46,A -85,B 0,C 180,E1 -2917.111,E2 -2917.111} C_VEL
LIN {X 0,Y 559.147,Z 268.461,A -85,B 0,C 180,E1 -2919.942,E2 -2919.942} C_VEL
LIN {X 0,Y 559.14,Z 268.457,A -85,B 0,C 180,E1 -2922.745,E2 -2922.745} C_VEL
LIN {X 0,Y 559.115,Z 268.465,A -85,B 0,C 180,E1 -2925.765,E2 -2925.765} C_VEL
LIN {X 0,Y 559.113,Z 268.465,A -85,B 0,C 180,E1 -2928.227,E2 -2928.227} C_VEL
LIN {X 0,Y 559.163,Z 268.454,A -85,B 0,C 180,E1 -2931.193,E2 -2931.193} C_VEL
LIN {X 0,Y 559.112,Z 268.467,A -85,B 0,C 180,E1 -2933.788,E2 -2933.788} C_VEL
LIN {X 0,Y 559.154,Z 268.457,A -85,B 0,C 180,E1 -2936.426,E2 -2936.426} C_VEL
LIN {X 0,Y 559.148,Z 268.455,A -85,B 0,C 180,E1 -2938.981,E2 -2938.981} C_VEL
LIN {X 0,Y 559.13,Z 268.466,A -85,B 0,C 180,E1 -2941.626,E2 -2941.626} C_VEL
LIN {X 0,Y 559.138,Z 268.618,A -85,B 0,C 180,E1 -2943.212,E2 -2943.212} C_VEL
LIN {X 0,Y 560.89,Z 276.344,A -85,B 0,C 180,E1 -2944.274,E2 -2944.274} C_VEL
LIN {X 0,Y 560.674,Z 294.608,A -85,B 0,C 180,E1 -2946.549,E2 -2946.549} C_VEL
LIN {X 0,Y 560.291,Z 316.685,A -85,B 0,C 180,E1 -2949.247,E2 -2949.247} C_VEL
LIN {X 0,Y 560.267,Z 322.113,A -85,B 0,C 180,E1 -2949.892,E2 -2949.892} C_VEL
LIN {X 0,Y 561.823,Z 330.817,A -85,B 0,C 180,E1 -2950.066,E2 -2950.066} C_VEL
LIN {X 0,Y 561.248,Z 488.117,A -85,B 0,C 180,E1 -2952.148,E2 -2952.148} C_VEL
LIN {X 0,Y 561.06,Z 503.72,A -85,B 0,C 180,E1 -2952.505,E2 -2952.505} C_VEL
LIN {X 0,Y 560.814,Z 519.048,A -85,B 0,C 180,E1 -2953.014,E2 -2953.014} C_VEL
LIN {X 0,Y 560.606,Z 532.787,A -85,B 0,C 180,E1 -2953.617,E2 -2953.617} C_VEL
LIN {X 0,Y 560.286,Z 546.258,A -85,B 0,C 180,E1 -2954.355,E2 -2954.355} C_VEL
LIN {X 0,Y 559.997,Z 559.308,A -85,B 0,C 180,E1 -2955.23,E2 -2955.23} C_VEL
LIN {X 0,Y 559.722,Z 571.297,A -85,B 0,C 180,E1 -2956.198,E2 -2956.198} C_VEL
LIN {X 0,Y 559.516,Z 582.753,A -85,B 0,C 180,E1 -2957.302,E2 -2957.302} C_VEL
LIN {X 0,Y 559.303,Z 592.392,A -85,B 0,C 180,E1 -2958.402,E2 -2958.402} C_VEL
LIN {X 0,Y 559.168,Z 601.857,A -85,B 0,C 180,E1 -2959.683,E2 -2959.683} C_VEL
LIN {X 0,Y 559.003,Z 609.737,A -85,B 0,C 180,E1 -2960.958,E2 -2960.958} C_VEL
LIN {X 0,Y 558.92,Z 617.091,A -85,B 0,C 180,E1 -2962.413,E2 -2962.413} C_VEL
LIN {X 0,Y 558.858,Z 622.923,A -85,B 0,C 180,E1 -2963.864,E2 -2963.864} C_VEL
LIN {X 0,Y 558.787,Z 626.387,A -85,B 0,C 180,E1 -2964.949,E2 -2964.949} C_VEL
LIN {X 0,Y 558.818,Z 629.889,A -85,B 0,C 180,E1 -2966.395,E2 -2966.395} C_VEL
LIN {X 0,Y 558.744,Z 632.191,A -85,B 0,C 180,E1 -2967.838,E2 -2967.838} C_VEL
LIN {X 0,Y 558.739,Z 633.349,A -85,B 0,C 180,E1 -2969.279,E2 -2969.279} C_VEL
LIN {X 0,Y 558.739,Z 633.348,A -85,B 0,C 180,E1 -2970.721,E2 -2970.721} C_VEL
LIN {X 0,Y 558.743,Z 632.189,A -85,B 0,C 180,E1 -2972.162,E2 -2972.162} C_VEL
LIN {X 0,Y 558.818,Z 629.886,A -85,B 0,C 180,E1 -2973.605,E2 -2973.605} C_VEL
LIN {X 0,Y 558.787,Z 626.387,A -85,B 0,C 180,E1 -2975.051,E2 -2975.051} C_VEL
LIN {X 0,Y 558.842,Z 621.609,A -85,B 0,C 180,E1 -2976.499,E2 -2976.499} C_VEL
LIN {X 0,Y 558.95,Z 615.423,A -85,B 0,C 180,E1 -2977.95,E2 -2977.95} C_VEL
LIN {X 0,Y 559.005,Z 607.647,A -85,B 0,C 180,E1 -2979.406,E2 -2979.406} C_VEL
LIN {X 0,Y 559.217,Z 599.37,A -85,B 0,C 180,E1 -2980.682,E2 -2980.682} C_VEL
LIN {X 0,Y 559.362,Z 589.394,A -85,B 0,C 180,E1 -2981.964,E2 -2981.964} C_VEL
LIN {X 0,Y 559.596,Z 579.19,A -85,B 0,C 180,E1 -2983.065,E2 -2983.065} C_VEL
LIN {X 0,Y 559.861,Z 567.024,A -85,B 0,C 180,E1 -2984.169,E2 -2984.169} C_VEL
LIN {X 0,Y 560.122,Z 554.693,A -85,B 0,C 180,E1 -2985.099,E2 -2985.099} C_VEL
LIN {X 0,Y 560.36,Z 541.517,A -85,B 0,C 180,E1 -2985.923,E2 -2985.923} C_VEL
LIN {X 0,Y 560.655,Z 526.835,A -85,B 0,C 180,E1 -2986.663,E2 -2986.663} C_VEL
LIN {X 0,Y 560.924,Z 512.628,A -85,B 0,C 180,E1 -2987.217,E2 -2987.217} C_VEL
LIN {X 0,Y 561.142,Z 498.161,A -85,B 0,C 180,E1 -2987.637,E2 -2987.637} C_VEL
LIN {X 0,Y 561.233,Z 483.666,A -85,B 0,C 180,E1 -2987.923,E2 -2987.923} C_VEL
LIN {X 0,Y 561.825,Z 330.818,A -85,B 0,C 180,E1 -2989.934,E2 -2989.934} C_VEL
LIN {X 0,Y 560.24,Z 321.913,A -85,B 0,C 180,E1 -2990.113,E2 -2990.113} C_VEL
LIN {X 0,Y 560.673,Z 296.183,A -85,B 0,C 180,E1 -2993.256,E2 -2993.256} C_VEL
LIN {X 0,Y 560.968,Z 277.544,A -85,B 0,C 180,E1 -2995.572,E2 -2995.572} C_VEL
LIN {X 0,Y 560.091,Z 272.497,A -85,B 0,C 180,E1 -2996.251,E2 -2996.251} C_VEL
LIN {X 0,Y 559.111,Z 268.466,A -85,B 0,C 180,E1 -2996.815,E2 -2996.815} C_VEL
LIN {X 0,Y 559.143,Z 268.462,A -85,B 0,C 180,E1 -2999.856,E2 -2999.856} C_VEL
LIN {X 0,Y 559.148,Z 268.457,A -85,B 0,C 180,E1 -3002.715,E2 -3002.715} C_VEL
LIN {X 0,Y 559.112,Z 268.46,A -85,B 0,C 180,E1 -3005.324,E2 -3005.324} C_VEL
LIN {X 0,Y 559.119,Z 268.468,A -85,B 0,C 180,E1 -3008.017,E2 -3008.017} C_VEL
LIN {X 0,Y 559.152,Z 268.463,A -85,B 0,C 180,E1 -3009.941,E2 -3009.941} C_VEL
LIN {X 0,Y 559.132,Z 268.458,A -85,B 0,C 180,E1 -3012.745,E2 -3012.745} C_VEL
LIN {X 0,Y 559.116,Z 268.466,A -85,B 0,C 180,E1 -3015.763,E2 -3015.763} C_VEL
LIN {X 0,Y 559.118,Z 268.464,A -85,B 0,C 180,E1 -3018.226,E2 -3018.226} C_VEL
LIN {X 0,Y 559.158,Z 268.454,A -85,B 0,C 180,E1 -3021.192,E2 -3021.192} C_VEL
LIN {X 0,Y 559.102,Z 268.469,A -85,B 0,C 180,E1 -3023.787,E2 -3023.787} C_VEL
LIN {X 0,Y 559.134,Z 268.458,A -85,B 0,C 180,E1 -3026.423,E2 -3026.423} C_VEL
LIN {X 0,Y 559.137,Z 268.456,A -85,B 0,C 180,E1 -3028.98,E2 -3028.98} C_VEL
LIN {X 0,Y 559.12,Z 268.466,A -85,B 0,C 180,E1 -3031.625,E2 -3031.625} C_VEL
LIN {X 0,Y 559.124,Z 268.458,A -85,B 0,C 180,E1 -3034.822,E2 -3034.822} C_VEL
LIN {X 0,Y 559.123,Z 268.465,A -85,B 0,C 180,E1 -3037.846,E2 -3037.846} C_VEL
LIN {X 0,Y 559.178,Z 268.447,A -85,B 0,C 180,E1 -3040.494,E2 -3040.494} C_VEL
LIN {X 0,Y 559.128,Z 268.459,A -85,B 0,C 180,E1 -3043.196,E2 -3043.196} C_VEL
LIN {X 0,Y 559.13,Z 268.457,A -85,B 0,C 180,E1 -3046.183,E2 -3046.183} C_VEL
LIN {X 0,Y 559.142,Z 268.453,A -85,B 0,C 180,E1 -3049.133,E2 -3049.133} C_VEL
LIN {X 0,Y 559.121,Z 268.46,A -85,B 0,C 180,E1 -3052.053,E2 -3052.053} C_VEL
LIN {X 0,Y 559.188,Z 268.449,A -85,B 0,C 180,E1 -3054.229,E2 -3054.229} C_VEL
LIN {X 0,Y 559.211,Z 268.452,A -85,B 0,C 180,E1 -3057.119,E2 -3057.119} C_VEL
LIN {X 0,Y 559.226,Z 268.447,A -85,B 0,C 180,E1 -3060,E2 -3060} C_VEL
LIN {X 0,Y 559.21,Z 268.449,A -85,B 0,C 180,E1 -3062.882,E2 -3062.882} C_VEL
LIN {X 0,Y 559.202,Z 268.45,A -85,B 0,C 180,E1 -3065.771,E2 -3065.771} C_VEL
LIN {X 0,Y 559.144,Z 268.457,A -85,B 0,C 180,E1 -3068.675,E2 -3068.675} C_VEL
LIN {X 0,Y 559.19,Z 268.453,A -85,B 0,C 180,E1 -3071.601,E2 -3071.601} C_VEL
LIN {X 0,Y 559.14,Z 268.457,A -85,B 0,C 180,E1 -3074.578,E2 -3074.578} C_VEL
LIN {X 0,Y 559.123,Z 268.461,A -85,B 0,C 180,E1 -3077.558,E2 -3077.558} C_VEL
LIN {X 0,Y 559.15,Z 268.451,A -85,B 0,C 180,E1 -3079.838,E2 -3079.838} C_VEL
LIN {X 0,Y 559.121,Z 268.456,A -85,B 0,C 180,E1 -3082.154,E2 -3082.154} C_VEL
LIN {X 0,Y 559.13,Z 268.463,A -85,B 0,C 180,E1 -3085.179,E2 -3085.179} C_VEL
LIN {X 0,Y 559.137,Z 268.454,A -85,B 0,C 180,E1 -3087.715,E2 -3087.715} C_VEL
LIN {X 0,Y 559.126,Z 268.46,A -85,B 0,C 180,E1 -3090.582,E2 -3090.582} C_VEL
LIN {X 0,Y 558.464,Z 268.548,A -85,B 0,C 180,E1 -3091.183,E2 -3091.183} C_VEL
LIN {X 0,Y 555.602,Z 268.904,A -85,B 0,C 180,E1 -3092.159,E2 -3092.159} C_VEL
LIN {X 0,Y 553.185,Z 269.207,A -85,B 0,C 180,E1 -3092.945,E2 -3092.945} C_VEL
LIN {X 0,Y 552.157,Z 269.328,A -85,B 0,C 180,E1 -3093.551,E2 -3093.551} C_VEL
LIN {X 0,Y 552.079,Z 269.336,A -85,B 0,C 180,E1 -3093.757,E2 -3093.757} C_VEL
LIN {X 0,Y 552.096,Z 269.341,A -85,B 0,C 180,E1 -3096.748,E2 -3096.748} C_VEL
LIN {X 0,Y 552.12,Z 269.331,A -85,B 0,C 180,E1 -3099.528,E2 -3099.528} C_VEL
LIN {X 0,Y 552.122,Z 269.334,A -85,B 0,C 180,E1 -3102.426,E2 -3102.426} C_VEL
LIN {X 0,Y 552.084,Z 269.336,A -85,B 0,C 180,E1 -3105.563,E2 -3105.563} C_VEL
LIN {X 0,Y 552.114,Z 269.339,A -85,B 0,C 180,E1 -3108.555,E2 -3108.555} C_VEL
LIN {X 0,Y 552.11,Z 269.332,A -85,B 0,C 180,E1 -3111.412,E2 -3111.412} C_VEL
LIN {X 0,Y 552.084,Z 269.337,A -85,B 0,C 180,E1 -3114.157,E2 -3114.157} C_VEL
LIN {X 0,Y 552.104,Z 269.34,A -85,B 0,C 180,E1 -3116.814,E2 -3116.814} C_VEL
LIN {X 0,Y 552.099,Z 269.335,A -85,B 0,C 180,E1 -3119.391,E2 -3119.391} C_VEL
LIN {X 0,Y 552.104,Z 269.335,A -85,B 0,C 180,E1 -3121.902,E2 -3121.902} C_VEL
LIN {X 0,Y 552.154,Z 269.335,A -85,B 0,C 180,E1 -3124.65,E2 -3124.65} C_VEL
LIN {X 0,Y 552.135,Z 269.531,A -85,B 0,C 180,E1 -3126.156,E2 -3126.156} C_VEL
LIN {X 0,Y 553.419,Z 276.213,A -85,B 0,C 180,E1 -3127.212,E2 -3127.212} C_VEL
LIN {X 0,Y 553.177,Z 293.337,A -85,B 0,C 180,E1 -3129.681,E2 -3129.681} C_VEL
LIN {X 0,Y 555.131,Z 303.6,A -85,B 0,C 180,E1 -3129.896,E2 -3129.896} C_VEL
LIN {X 0,Y 554.48,Z 458.351,A -85,B 0,C 180,E1 -3131.972,E2 -3131.972} C_VEL
LIN {X 0,Y 554.288,Z 473.824,A -85,B 0,C 180,E1 -3132.332,E2 -3132.332} C_VEL
LIN {X 0,Y 554.022,Z 489.116,A -85,B 0,C 180,E1 -3132.847,E2 -3132.847} C_VEL
LIN {X 0,Y 553.768,Z 501.846,A -85,B 0,C 180,E1 -3133.409,E2 -3133.409} C_VEL
LIN {X 0,Y 553.414,Z 515.507,A -85,B 0,C 180,E1 -3134.155,E2 -3134.155} C_VEL
LIN {X 0,Y 553.125,Z 528.083,A -85,B 0,C 180,E1 -3134.998,E2 -3134.998} C_VEL
LIN {X 0,Y 552.803,Z 540.788,A -85,B 0,C 180,E1 -3136.022,E2 -3136.022} C_VEL
LIN {X 0,Y 552.548,Z 552.322,A -85,B 0,C 180,E1 -3137.139,E2 -3137.139} C_VEL
LIN {X 0,Y 552.29,Z 562.033,A -85,B 0,C 180,E1 -3138.253,E2 -3138.253} C_VEL
LIN {X 0,Y 552.133,Z 571.556,A -85,B 0,C 180,E1 -3139.55,E2 -3139.55} C_VEL
LIN {X 0,Y 551.922,Z 580.493,A -85,B 0,C 180,E1 -3141.026,E2 -3141.026} C_VEL
LIN {X 0,Y 551.839,Z 586.892,A -85,B 0,C 180,E1 -3142.315,E2 -3142.315} C_VEL
LIN {X 0,Y 551.747,Z 592.496,A -85,B 0,C 180,E1 -3143.703,E2 -3143.703} C_VEL
LIN {X 0,Y 551.713,Z 596.257,A -85,B 0,C 180,E1 -3144.884,E2 -3144.884} C_VEL
LIN {X 0,Y 551.73,Z 599.796,A -85,B 0,C 180,E1 -3146.348,E2 -3146.348} C_VEL
LIN {X 0,Y 551.655,Z 602.138,A -85,B 0,C 180,E1 -3147.81,E2 -3147.81} C_VEL
LIN {X 0,Y 551.637,Z 603.337,A -85,B 0,C 180,E1 -3149.27,E2 -3149.27} C_VEL
LIN {X 0,Y 551.638,Z 603.358,A -85,B 0,C 180,E1 -3150.73,E2 -3150.73} C_VEL
LIN {X 0,Y 551.655,Z 602.24,A -85,B 0,C 180,E1 -3152.19,E2 -3152.19} C_VEL
LIN {X 0,Y 551.732,Z 599.978,A -85,B 0,C 180,E1 -3153.652,E2 -3153.652} C_VEL
LIN {X 0,Y 551.712,Z 596.517,A -85,B 0,C 180,E1 -3155.116,E2 -3155.116} C_VEL
LIN {X 0,Y 551.781,Z 591.781,A -85,B 0,C 180,E1 -3156.582,E2 -3156.582} C_VEL
LIN {X 0,Y 551.877,Z 585.645,A -85,B 0,C 180,E1 -3158.052,E2 -3158.052} C_VEL
LIN {X 0,Y 551.949,Z 577.922,A -85,B 0,C 180,E1 -3159.528,E2 -3159.528} C_VEL
LIN {X 0,Y 552.168,Z 569.685,A -85,B 0,C 180,E1 -3160.821,E2 -3160.821} C_VEL
LIN {X 0,Y 552.344,Z 559.773,A -85,B 0,C 180,E1 -3162.119,E2 -3162.119} C_VEL
LIN {X 0,Y 552.593,Z 549.616,A -85,B 0,C 180,E1 -3163.234,E2 -3163.234} C_VEL
LIN {X 0,Y 552.88,Z 537.53,A -85,B 0,C 180,E1 -3164.351,E2 -3164.351} C_VEL
LIN {X 0,Y 553.235,Z 524.858,A -85,B 0,C 180,E1 -3165.324,E2 -3165.324} C_VEL
LIN {X 0,Y 553.521,Z 512.271,A -85,B 0,C 180,E1 -3166.125,E2 -3166.125} C_VEL
LIN {X 0,Y 553.801,Z 499.762,A -85,B 0,C 180,E1 -3166.78,E2 -3166.78} C_VEL
LIN {X 0,Y 554.112,Z 485.142,A -85,B 0,C 180,E1 -3167.388,E2 -3167.388} C_VEL
LIN {X 0,Y 554.336,Z 469.545,A -85,B 0,C 180,E1 -3167.869,E2 -3167.869} C_VEL
LIN {X 0,Y 554.492,Z 454.499,A -85,B 0,C 180,E1 -3168.18,E2 -3168.18} C_VEL
LIN {X 0,Y 555.133,Z 303.28,A -85,B 0,C 180,E1 -3170.198,E2 -3170.198} C_VEL
LIN {X 0,Y 553.094,Z 292.973,A -85,B 0,C 180,E1 -3170.438,E2 -3170.438} C_VEL
LIN {X 0,Y 553.461,Z 276.851,A -85,B 0,C 180,E1 -3172.786,E2 -3172.786} C_VEL
LIN {X 0,Y 552.15,Z 269.335,A -85,B 0,C 180,E1 -3173.974,E2 -3173.974} C_VEL
LIN {X 0,Y 552.118,Z 269.332,A -85,B 0,C 180,E1 -3176.456,E2 -3176.456} C_VEL
LIN {X 0,Y 552.097,Z 269.337,A -85,B 0,C 180,E1 -3178.928,E2 -3178.928} C_VEL
LIN {X 0,Y 552.108,Z 269.342,A -85,B 0,C 180,E1 -3181.475,E2 -3181.475} C_VEL
LIN {X 0,Y 552.134,Z 269.33,A -85,B 0,C 180,E1 -3184.17,E2 -3184.17} C_VEL
LIN {X 0,Y 552.105,Z 269.335,A -85,B 0,C 180,E1 -3186.746,E2 -3186.746} C_VEL
LIN {X 0,Y 552.127,Z 269.335,A -85,B 0,C 180,E1 -3189.526,E2 -3189.526} C_VEL
LIN {X 0,Y 552.124,Z 269.331,A -85,B 0,C 180,E1 -3192.425,E2 -3192.425} C_VEL
LIN {X 0,Y 552.084,Z 269.34,A -85,B 0,C 180,E1 -3195.561,E2 -3195.561} C_VEL
LIN {X 0,Y 552.113,Z 269.329,A -85,B 0,C 180,E1 -3198.553,E2 -3198.553} C_VEL
LIN {X 0,Y 552.107,Z 269.337,A -85,B 0,C 180,E1 -3201.41,E2 -3201.41} C_VEL
LIN {X 0,Y 552.077,Z 269.333,A -85,B 0,C 180,E1 -3204.156,E2 -3204.156} C_VEL
LIN {X 0,Y 552.097,Z 269.338,A -85,B 0,C 180,E1 -3206.813,E2 -3206.813} C_VEL
LIN {X 0,Y 552.091,Z 269.335,A -85,B 0,C 180,E1 -3209.39,E2 -3209.39} C_VEL
LIN {X 0,Y 552.085,Z 269.335,A -85,B 0,C 180,E1 -3211.9,E2 -3211.9} C_VEL
LIN {X 0,Y 552.096,Z 269.337,A -85,B 0,C 180,E1 -3214.66,E2 -3214.66} C_VEL
LIN {X 0,Y 552.075,Z 269.337,A -85,B 0,C 180,E1 -3217.548,E2 -3217.548} C_VEL
LIN {X 0,Y 552.131,Z 269.331,A -85,B 0,C 180,E1 -3220.375,E2 -3220.375} C_VEL
LIN {X 0,Y 552.141,Z 269.336,A -85,B 0,C 180,E1 -3222.977,E2 -3222.977} C_VEL
LIN {X 0,Y 552.108,Z 269.331,A -85,B 0,C 180,E1 -3226.004,E2 -3226.004} C_VEL
LIN {X 0,Y 552.138,Z 269.335,A -85,B 0,C 180,E1 -3228.993,E2 -3228.993} C_VEL
LIN {X 0,Y 552.13,Z 269.328,A -85,B 0,C 180,E1 -3231.951,E2 -3231.951} C_VEL
LIN {X 0,Y 552.202,Z 269.325,A -85,B 0,C 180,E1 -3234.889,E2 -3234.889} C_VEL
LIN {X 0,Y 552.194,Z 269.321,A -85,B 0,C 180,E1 -3237.812,E2 -3237.812} C_VEL
LIN {X 0,Y 552.23,Z 269.325,A -85,B 0,C 180,E1 -3240.729,E2 -3240.729} C_VEL
LIN {X 0,Y 552.178,Z 269.327,A -85,B 0,C 180,E1 -3242.918,E2 -3242.918} C_VEL
LIN {X 0,Y 552.162,Z 269.325,A -85,B 0,C 180,E1 -3245.844,E2 -3245.844} C_VEL
LIN {X 0,Y 552.113,Z 269.336,A -85,B 0,C 180,E1 -3248.786,E2 -3248.786} C_VEL
LIN {X 0,Y 552.142,Z 269.329,A -85,B 0,C 180,E1 -3251.751,E2 -3251.751} C_VEL
LIN {X 0,Y 552.12,Z 269.336,A -85,B 0,C 180,E1 -3254.749,E2 -3254.749} C_VEL
LIN {X 0,Y 552.068,Z 269.337,A -85,B 0,C 180,E1 -3257.79,E2 -3257.79} C_VEL
LIN {X 0,Y 552.11,Z 269.337,A -85,B 0,C 180,E1 -3260.102,E2 -3260.102} C_VEL
LIN {X 0,Y 552.074,Z 269.345,A -85,B 0,C 180,E1 -3262.452,E2 -3262.452} C_VEL
LIN {X 0,Y 552.065,Z 269.337,A -85,B 0,C 180,E1 -3265.334,E2 -3265.334} C_VEL
LIN {X 0,Y 552.063,Z 269.345,A -85,B 0,C 180,E1 -3268.101,E2 -3268.101} C_VEL
LIN {X 0,Y 552.08,Z 269.339,A -85,B 0,C 180,E1 -3270.611,E2 -3270.611} C_VEL
LIN {X 0,Y 552.093,Z 269.332,A -85,B 0,C 180,E1 -3273.187,E2 -3273.187} C_VEL
LIN {X 0,Y 552.057,Z 269.343,A -85,B 0,C 180,E1 -3275.846,E2 -3275.846} C_VEL
LIN {X 0,Y 552.105,Z 269.331,A -85,B 0,C 180,E1 -3279.061,E2 -3279.061} C_VEL
LIN {X 0,Y 552.069,Z 269.335,A -85,B 0,C 180,E1 -3281.451,E2 -3281.451} C_VEL
LIN {X 0,Y 552.066,Z 269.341,A -85,B 0,C 180,E1 -3284.441,E2 -3284.441} C_VEL
LIN {X 0,Y 552.078,Z 269.339,A -85,B 0,C 180,E1 -3287.591,E2 -3287.591} C_VEL
LIN {X 0,Y 552.12,Z 269.333,A -85,B 0,C 180,E1 -3290.473,E2 -3290.473} C_VEL
LIN {X 0,Y 552.091,Z 269.336,A -85,B 0,C 180,E1 -3293.319,E2 -3293.319} C_VEL
LIN {X 0,Y 552.118,Z 269.34,A -85,B 0,C 180,E1 -3295.94,E2 -3295.94} C_VEL
LIN {X 0,Y 552.115,Z 269.332,A -85,B 0,C 180,E1 -3298.541,E2 -3298.541} C_VEL
LIN {X 0,Y 552.093,Z 269.341,A -85,B 0,C 180,E1 -3301.444,E2 -3301.444} C_VEL
LIN {X 0,Y 552.098,Z 269.431,A -85,B 0,C 180,E1 -3302.973,E2 -3302.973} C_VEL
LIN {X 0,Y 554.088,Z 278.475,A -85,B 0,C 180,E1 -3304.231,E2 -3304.231} C_VEL
LIN {X 0,Y 553.78,Z 297.57,A -85,B 0,C 180,E1 -3306.635,E2 -3306.635} C_VEL
LIN {X 0,Y 553.34,Z 321.716,A -85,B 0,C 180,E1 -3309.616,E2 -3309.616} C_VEL
LIN {X 0,Y 555.156,Z 332.094,A -85,B 0,C 180,E1 -3309.834,E2 -3309.834} C_VEL
LIN {X 0,Y 554.484,Z 487.813,A -85,B 0,C 180,E1 -3311.918,E2 -3311.918} C_VEL
LIN {X 0,Y 554.307,Z 503.718,A -85,B 0,C 180,E1 -3312.285,E2 -3312.285} C_VEL
LIN {X 0,Y 554.014,Z 519.045,A -85,B 0,C 180,E1 -3312.799,E2 -3312.799} C_VEL
LIN {X 0,Y 553.773,Z 532.79,A -85,B 0,C 180,E1 -3313.409,E2 -3313.409} C_VEL
LIN {X 0,Y 553.405,Z 546.26,A -85,B 0,C 180,E1 -3314.155,E2 -3314.155} C_VEL
LIN {X 0,Y 553.077,Z 560.15,A -85,B 0,C 180,E1 -3315.103,E2 -3315.103} C_VEL
LIN {X 0,Y 552.76,Z 572.358,A -85,B 0,C 180,E1 -3316.115,E2 -3316.115} C_VEL
LIN {X 0,Y 552.482,Z 584.512,A -85,B 0,C 180,E1 -3317.325,E2 -3317.325} C_VEL
LIN {X 0,Y 552.215,Z 594.486,A -85,B 0,C 180,E1 -3318.514,E2 -3318.514} C_VEL
LIN {X 0,Y 552.124,Z 603.088,A -85,B 0,C 180,E1 -3319.735,E2 -3319.735} C_VEL
LIN {X 0,Y 551.921,Z 610.744,A -85,B 0,C 180,E1 -3321.026,E2 -3321.026} C_VEL
LIN {X 0,Y 551.837,Z 617.091,A -85,B 0,C 180,E1 -3322.315,E2 -3322.315} C_VEL
LIN {X 0,Y 551.758,Z 622.608,A -85,B 0,C 180,E1 -3323.692,E2 -3323.692} C_VEL
LIN {X 0,Y 551.713,Z 626.387,A -85,B 0,C 180,E1 -3324.884,E2 -3324.884} C_VEL
LIN {X 0,Y 551.73,Z 629.888,A -85,B 0,C 180,E1 -3326.348,E2 -3326.348} C_VEL
LIN {X 0,Y 551.654,Z 632.19,A -85,B 0,C 180,E1 -3327.81,E2 -3327.81} C_VEL
LIN {X 0,Y 551.639,Z 633.348,A -85,B 0,C 180,E1 -3329.27,E2 -3329.27} C_VEL
LIN {X 0,Y 551.639,Z 633.348,A -85,B 0,C 180,E1 -3330.73,E2 -3330.73} C_VEL
LIN {X 0,Y 551.654,Z 632.188,A -85,B 0,C 180,E1 -3332.19,E2 -3332.19} C_VEL
LIN {X 0,Y 551.73,Z 629.885,A -85,B 0,C 180,E1 -3333.652,E2 -3333.652} C_VEL
LIN {X 0,Y 551.713,Z 626.387,A -85,B 0,C 180,E1 -3335.116,E2 -3335.116} C_VEL
LIN {X 0,Y 551.779,Z 621.61,A -85,B 0,C 180,E1 -3336.582,E2 -3336.582} C_VEL
LIN {X 0,Y 551.876,Z 615.422,A -85,B 0,C 180,E1 -3338.052,E2 -3338.052} C_VEL
LIN {X 0,Y 551.95,Z 607.646,A -85,B 0,C 180,E1 -3339.528,E2 -3339.528} C_VEL
LIN {X 0,Y 552.184,Z 599.37,A -85,B 0,C 180,E1 -3340.82,E2 -3340.82} C_VEL
LIN {X 0,Y 552.352,Z 589.394,A -85,B 0,C 180,E1 -3342.119,E2 -3342.119} C_VEL
LIN {X 0,Y 552.609,Z 579.189,A -85,B 0,C 180,E1 -3343.233,E2 -3343.233} C_VEL
LIN {X 0,Y 552.906,Z 567.024,A -85,B 0,C 180,E1 -3344.351,E2 -3344.351} C_VEL
LIN {X 0,Y 553.242,Z 554.447,A -85,B 0,C 180,E1 -3345.31,E2 -3345.31} C_VEL
LIN {X 0,Y 553.51,Z 541.514,A -85,B 0,C 180,E1 -3346.125,E2 -3346.125} C_VEL
LIN {X 0,Y 553.847,Z 526.833,A -85,B 0,C 180,E1 -3346.874,E2 -3346.874} C_VEL
LIN {X 0,Y 554.141,Z 512.628,A -85,B 0,C 180,E1 -3347.435,E2 -3347.435} C_VEL
LIN {X 0,Y 554.398,Z 497.523,A -85,B 0,C 180,E1 -3347.875,E2 -3347.875} C_VEL
LIN {X 0,Y 554.504,Z 483.332,A -85,B 0,C 180,E1 -3348.153,E2 -3348.153} C_VEL
LIN {X 0,Y 555.14,Z 331.349,A -85,B 0,C 180,E1 -3350.177,E2 -3350.177} C_VEL
LIN {X 0,Y 553.348,Z 321.705,A -85,B 0,C 180,E1 -3350.385,E2 -3350.385} C_VEL
LIN {X 0,Y 553.784,Z 297.569,A -85,B 0,C 180,E1 -3353.364,E2 -3353.364} C_VEL
LIN {X 0,Y 554.117,Z 280.226,A -85,B 0,C 180,E1 -3355.545,E2 -3355.545} C_VEL
LIN {X 0,Y 553.821,Z 276.71,A -85,B 0,C 180,E1 -3356.008,E2 -3356.008} C_VEL
LIN {X 0,Y 552.078,Z 269.342,A -85,B 0,C 180,E1 -3357.048,E2 -3357.048} C_VEL
LIN {X 0,Y 552.111,Z 269.339,A -85,B 0,C 180,E1 -3360.05,E2 -3360.05} C_VEL
LIN {X 0,Y 552.107,Z 269.334,A -85,B 0,C 180,E1 -3362.845,E2 -3362.845} C_VEL
LIN {X 0,Y 552.06,Z 269.339,A -85,B 0,C 180,E1 -3365.437,E2 -3365.437} C_VEL
LIN {X 0,Y 552.083,Z 269.342,A -85,B 0,C 180,E1 -3367.884,E2 -3367.884} C_VEL
LIN {X 0,Y 552.085,Z 269.339,A -85,B 0,C 180,E1 -3370.482,E2 -3370.482} C_VEL
LIN {X 0,Y 552.056,Z 269.341,A -85,B 0,C 180,E1 -3373.478,E2 -3373.478} C_VEL
LIN {X 0,Y 552.063,Z 269.339,A -85,B 0,C 180,E1 -3376.572,E2 -3376.572} C_VEL
LIN {X 0,Y 552.082,Z 269.339,A -85,B 0,C 180,E1 -3379.517,E2 -3379.517} C_VEL
LIN {X 0,Y 552.071,Z 269.339,A -85,B 0,C 180,E1 -3382.335,E2 -3382.335} C_VEL
LIN {X 0,Y 552.061,Z 269.337,A -85,B 0,C 180,E1 -3385.049,E2 -3385.049} C_VEL
LIN {X 0,Y 552.101,Z 269.34,A -85,B 0,C 180,E1 -3387.68,E2 -3387.68} C_VEL
LIN {X 0,Y 552.072,Z 269.339,A -85,B 0,C 180,E1 -3390.233,E2 -3390.233} C_VEL
LIN {X 0,Y 552.065,Z 269.337,A -85,B 0,C 180,E1 -3393.012,E2 -3393.012} C_VEL
LIN {X 0,Y 552.067,Z 269.342,A -85,B 0,C 180,E1 -3395.96,E2 -3395.96} C_VEL
LIN {X 0,Y 552.101,Z 269.334,A -85,B 0,C 180,E1 -3399.119,E2 -3399.119} C_VEL
LIN {X 0,Y 552.067,Z 269.339,A -85,B 0,C 180,E1 -3401.442,E2 -3401.442} C_VEL
LIN {X 0,Y 552.072,Z 269.344,A -85,B 0,C 180,E1 -3403.736,E2 -3403.736} C_VEL
LIN {X 0,Y 552.097,Z 269.335,A -85,B 0,C 180,E1 -3406.004,E2 -3406.004} C_VEL
LIN {X 0,Y 552.105,Z 269.327,A -85,B 0,C 180,E1 -3408.992,E2 -3408.992} C_VEL
LIN {X 0,Y 552.091,Z 269.337,A -85,B 0,C 180,E1 -3411.951,E2 -3411.951} C_VEL
LIN {X 0,Y 552.161,Z 269.324,A -85,B 0,C 180,E1 -3414.156,E2 -3414.156} C_VEL
LIN {X 0,Y 552.176,Z 269.328,A -85,B 0,C 180,E1 -3417.082,E2 -3417.082} C_VEL
LIN {X 0,Y 552.196,Z 269.322,A -85,B 0,C 180,E1 -3420,E2 -3420} C_VEL
LIN {X 0,Y 552.178,Z 269.325,A -85,B 0,C 180,E1 -3422.918,E2 -3422.918} C_VEL
LIN {X 0,Y 552.17,Z 269.325,A -85,B 0,C 180,E1 -3425.844,E2 -3425.844} C_VEL
LIN {X 0,Y 552.117,Z 269.333,A -85,B 0,C 180,E1 -3428.786,E2 -3428.786} C_VEL
LIN {X 0,Y 552.146,Z 269.329,A -85,B 0,C 180,E1 -3431.751,E2 -3431.751} C_VEL
LIN {X 0,Y 552.106,Z 269.335,A -85,B 0,C 180,E1 -3434.749,E2 -3434.749} C_VEL
LIN {X 0,Y 552.081,Z 269.336,A -85,B 0,C 180,E1 -3437.79,E2 -3437.79} C_VEL
LIN {X 0,Y 552.111,Z 269.326,A -85,B 0,C 180,E1 -3440.102,E2 -3440.102} C_VEL
LIN {X 0,Y 552.073,Z 269.335,A -85,B 0,C 180,E1 -3442.452,E2 -3442.452} C_VEL
LIN {X 0,Y 552.099,Z 269.333,A -85,B 0,C 180,E1 -3445.646,E2 -3445.646} C_VEL
LIN {X 0,Y 552.081,Z 269.332,A -85,B 0,C 180,E1 -3448.1,E2 -3448.1} C_VEL
LIN {X 0,Y 552.09,Z 269.338,A -85,B 0,C 180,E1 -3450.61,E2 -3450.61} C_VEL
LIN {X 0,Y 552.095,Z 269.339,A -85,B 0,C 180,E1 -3453.187,E2 -3453.187} C_VEL
LIN {X 0,Y 552.079,Z 269.336,A -85,B 0,C 180,E1 -3453.757,E2 -3453.757} C_VEL
LIN {X 0,Y 551.438,Z 269.418,A -85,B 0,C 180,E1 -3454.365,E2 -3454.365} C_VEL
LIN {X 0,Y 548.628,Z 269.775,A -85,B 0,C 180,E1 -3455.354,E2 -3455.354} C_VEL
LIN {X 0,Y 546.222,Z 270.079,A -85,B 0,C 180,E1 -3456.15,E2 -3456.15} C_VEL
LIN {X 0,Y 545.158,Z 270.208,A -85,B 0,C 180,E1 -3456.763,E2 -3456.763} C_VEL
LIN {X 0,Y 545.055,Z 270.217,A -85,B 0,C 180,E1 -3456.971,E2 -3456.971} C_VEL
LIN {X 0,Y 545.056,Z 270.21,A -85,B 0,C 180,E1 -3460.144,E2 -3460.144} C_VEL
LIN {X 0,Y 545.071,Z 270.214,A -85,B 0,C 180,E1 -3463.107,E2 -3463.107} C_VEL
LIN {X 0,Y 545.042,Z 270.215,A -85,B 0,C 180,E1 -3466.227,E2 -3466.227} C_VEL
LIN {X 0,Y 545.075,Z 270.216,A -85,B 0,C 180,E1 -3468.886,E2 -3468.886} C_VEL
LIN {X 0,Y 545.073,Z 270.214,A -85,B 0,C 180,E1 -3470.819,E2 -3470.819} C_VEL
LIN {X 0,Y 545.039,Z 270.212,A -85,B 0,C 180,E1 -3473.621,E2 -3473.621} C_VEL
LIN {X 0,Y 545.048,Z 270.217,A -85,B 0,C 180,E1 -3476.328,E2 -3476.328} C_VEL
LIN {X 0,Y 545.063,Z 270.215,A -85,B 0,C 180,E1 -3478.953,E2 -3478.953} C_VEL
LIN {X 0,Y 545.082,Z 270.209,A -85,B 0,C 180,E1 -3481.507,E2 -3481.507} C_VEL
LIN {X 0,Y 545.093,Z 270.215,A -85,B 0,C 180,E1 -3484.492,E2 -3484.492} C_VEL
LIN {X 0,Y 545.106,Z 270.398,A -85,B 0,C 180,E1 -3485.931,E2 -3485.931} C_VEL
LIN {X 0,Y 546.549,Z 277.741,A -85,B 0,C 180,E1 -3487.11,E2 -3487.11} C_VEL
LIN {X 0,Y 546.241,Z 293.255,A -85,B 0,C 180,E1 -3489.399,E2 -3489.399} C_VEL
LIN {X 0,Y 548.481,Z 303.848,A -85,B 0,C 180,E1 -3489.641,E2 -3489.641} C_VEL
LIN {X 0,Y 547.743,Z 458.577,A -85,B 0,C 180,E1 -3491.743,E2 -3491.743} C_VEL
LIN {X 0,Y 547.526,Z 473.985,A -85,B 0,C 180,E1 -3492.106,E2 -3492.106} C_VEL
LIN {X 0,Y 547.249,Z 489.235,A -85,B 0,C 180,E1 -3492.628,E2 -3492.628} C_VEL
LIN {X 0,Y 546.956,Z 501.925,A -85,B 0,C 180,E1 -3493.196,E2 -3493.196} C_VEL
LIN {X 0,Y 546.55,Z 515.536,A -85,B 0,C 180,E1 -3493.951,E2 -3493.951} C_VEL
LIN {X 0,Y 546.21,Z 529.111,A -85,B 0,C 180,E1 -3494.879,E2 -3494.879} C_VEL
LIN {X 0,Y 545.874,Z 540.793,A -85,B 0,C 180,E1 -3495.841,E2 -3495.841} C_VEL
LIN {X 0,Y 545.572,Z 552.327,A -85,B 0,C 180,E1 -3496.972,E2 -3496.972} C_VEL
LIN {X 0,Y 545.289,Z 562.037,A -85,B 0,C 180,E1 -3498.1,E2 -3498.1} C_VEL
LIN {X 0,Y 545.09,Z 571.559,A -85,B 0,C 180,E1 -3499.413,E2 -3499.413} C_VEL
LIN {X 0,Y 544.877,Z 580.496,A -85,B 0,C 180,E1 -3500.909,E2 -3500.909} C_VEL
LIN {X 0,Y 544.773,Z 586.894,A -85,B 0,C 180,E1 -3502.215,E2 -3502.215} C_VEL
LIN {X 0,Y 544.676,Z 592.018,A -85,B 0,C 180,E1 -3503.483,E2 -3503.483} C_VEL
LIN {X 0,Y 544.642,Z 596.258,A -85,B 0,C 180,E1 -3504.818,E2 -3504.818} C_VEL
LIN {X 0,Y 544.645,Z 599.796,A -85,B 0,C 180,E1 -3506.301,E2 -3506.301} C_VEL
LIN {X 0,Y 544.569,Z 602.138,A -85,B 0,C 180,E1 -3507.781,E2 -3507.781} C_VEL
LIN {X 0,Y 544.537,Z 603.337,A -85,B 0,C 180,E1 -3509.261,E2 -3509.261} C_VEL
LIN {X 0,Y 544.538,Z 603.358,A -85,B 0,C 180,E1 -3510.739,E2 -3510.739} C_VEL
LIN {X 0,Y 544.57,Z 602.238,A -85,B 0,C 180,E1 -3512.219,E2 -3512.219} C_VEL
LIN {X 0,Y 544.646,Z 599.976,A -85,B 0,C 180,E1 -3513.699,E2 -3513.699} C_VEL
LIN {X 0,Y 544.641,Z 596.516,A -85,B 0,C 180,E1 -3515.182,E2 -3515.182} C_VEL
LIN {X 0,Y 544.698,Z 591.778,A -85,B 0,C 180,E1 -3516.668,E2 -3516.668} C_VEL
LIN {X 0,Y 544.819,Z 585.642,A -85,B 0,C 180,E1 -3518.157,E2 -3518.157} C_VEL
LIN {X 0,Y 544.903,Z 577.918,A -85,B 0,C 180,E1 -3519.652,E2 -3519.652} C_VEL
LIN {X 0,Y 545.128,Z 569.681,A -85,B 0,C 180,E1 -3520.962,E2 -3520.962} C_VEL
LIN {X 0,Y 545.332,Z 559.769,A -85,B 0,C 180,E1 -3522.277,E2 -3522.277} C_VEL
LIN {X 0,Y 545.617,Z 549.609,A -85,B 0,C 180,E1 -3523.406,E2 -3523.406} C_VEL
LIN {X 0,Y 545.922,Z 537.521,A -85,B 0,C 180,E1 -3524.538,E2 -3524.538} C_VEL
LIN {X 0,Y 546.329,Z 525.24,A -85,B 0,C 180,E1 -3525.494,E2 -3525.494} C_VEL
LIN {X 0,Y 546.676,Z 512.293,A -85,B 0,C 180,E1 -3526.333,E2 -3526.333} C_VEL
LIN {X 0,Y 547.004,Z 499.823,A -85,B 0,C 180,E1 -3526.995,E2 -3526.995} C_VEL
LIN {X 0,Y 547.319,Z 486.537,A -85,B 0,C 180,E1 -3527.563,E2 -3527.563} C_VEL
LIN {X 0,Y 547.562,Z 471.415,A -85,B 0,C 180,E1 -3528.052,E2 -3528.052} C_VEL
LIN {X 0,Y 547.71,Z 456.816,A -85,B 0,C 180,E1 -3528.378,E2 -3528.378} C_VEL
LIN {X 0,Y 548.469,Z 304.439,A -85,B 0,C 180,E1 -3530.441,E2 -3530.441} C_VEL
LIN {X 0,Y 546.251,Z 293.26,A -85,B 0,C 180,E1 -3530.693,E2 -3530.693} C_VEL
LIN {X 0,Y 546.606,Z 278.363,A -85,B 0,C 180,E1 -3532.888,E2 -3532.888} C_VEL
LIN {X 0,Y 545.089,Z 270.213,A -85,B 0,C 180,E1 -3534.205,E2 -3534.205} C_VEL
LIN {X 0,Y 545.091,Z 270.212,A -85,B 0,C 180,E1 -3537.173,E2 -3537.173} C_VEL
LIN {X 0,Y 545.075,Z 270.211,A -85,B 0,C 180,E1 -3540.246,E2 -3540.246} C_VEL
LIN {X 0,Y 545.077,Z 270.213,A -85,B 0,C 180,E1 -3543.062,E2 -3543.062} C_VEL
LIN {X 0,Y 545.05,Z 270.219,A -85,B 0,C 180,E1 -3545.675,E2 -3545.675} C_VEL
LIN {X 0,Y 545.047,Z 270.213,A -85,B 0,C 180,E1 -3548.236,E2 -3548.236} C_VEL
LIN {X 0,Y 545.076,Z 270.207,A -85,B 0,C 180,E1 -3550.472,E2 -3550.472} C_VEL
LIN {X 0,Y 545.072,Z 270.215,A -85,B 0,C 180,E1 -3553.106,E2 -3553.106} C_VEL
LIN {X 0,Y 545.042,Z 270.213,A -85,B 0,C 180,E1 -3556.225,E2 -3556.225} C_VEL
LIN {X 0,Y 545.073,Z 270.208,A -85,B 0,C 180,E1 -3558.884,E2 -3558.884} C_VEL
LIN {X 0,Y 545.07,Z 270.212,A -85,B 0,C 180,E1 -3560.817,E2 -3560.817} C_VEL
LIN {X 0,Y 545.033,Z 270.214,A -85,B 0,C 180,E1 -3563.619,E2 -3563.619} C_VEL
LIN {X 0,Y 545.041,Z 270.213,A -85,B 0,C 180,E1 -3566.326,E2 -3566.326} C_VEL
LIN {X 0,Y 545.055,Z 270.214,A -85,B 0,C 180,E1 -3568.951,E2 -3568.951} C_VEL
LIN {X 0,Y 545.072,Z 270.211,A -85,B 0,C 180,E1 -3571.506,E2 -3571.506} C_VEL
LIN {X 0,Y 545.058,Z 270.209,A -85,B 0,C 180,E1 -3573.998,E2 -3573.998} C_VEL
LIN {X 0,Y 545.02,Z 270.219,A -85,B 0,C 180,E1 -3577.241,E2 -3577.241} C_VEL
LIN {X 0,Y 545.103,Z 270.207,A -85,B 0,C 180,E1 -3580.414,E2 -3580.414} C_VEL
LIN {X 0,Y 545.054,Z 270.212,A -85,B 0,C 180,E1 -3583.52,E2 -3583.52} C_VEL
LIN {X 0,Y 545.07,Z 270.208,A -85,B 0,C 180,E1 -3585.819,E2 -3585.819} C_VEL
LIN {X 0,Y 545.097,Z 270.214,A -85,B 0,C 180,E1 -3588.849,E2 -3588.849} C_VEL
LIN {X 0,Y 545.078,Z 270.207,A -85,B 0,C 180,E1 -3591.846,E2 -3591.846} C_VEL
LIN {X 0,Y 545.179,Z 270.201,A -85,B 0,C 180,E1 -3594.823,E2 -3594.823} C_VEL
LIN {X 0,Y 545.167,Z 270.197,A -85,B 0,C 180,E1 -3597.783,E2 -3597.783} C_VEL
LIN {X 0,Y 545.199,Z 270.201,A -85,B 0,C 180,E1 -3600.739,E2 -3600.739} C_VEL
LIN {X 0,Y 545.143,Z 270.203,A -85,B 0,C 180,E1 -3602.956,E2 -3602.956} C_VEL
LIN {X 0,Y 545.114,Z 270.203,A -85,B 0,C 180,E1 -3605.92,E2 -3605.92} C_VEL
LIN {X 0,Y 545.05,Z 270.215,A -85,B 0,C 180,E1 -3608.154,E2 -3608.154} C_VEL
LIN {X 0,Y 545.096,Z 270.207,A -85,B 0,C 180,E1 -3611.151,E2 -3611.151} C_VEL
LIN {X 0,Y 545.074,Z 270.212,A -85,B 0,C 180,E1 -3614.181,E2 -3614.181} C_VEL
LIN {X 0,Y 545.042,Z 270.211,A -85,B 0,C 180,E1 -3617.416,E2 -3617.416} C_VEL
LIN {X 0,Y 545.076,Z 270.218,A -85,B 0,C 180,E1 -3620.373,E2 -3620.373} C_VEL
LIN {X 0,Y 545.059,Z 270.211,A -85,B 0,C 180,E1 -3623.56,E2 -3623.56} C_VEL
LIN {X 0,Y 545.022,Z 270.219,A -85,B 0,C 180,E1 -3626.003,E2 -3626.003} C_VEL
LIN {X 0,Y 545.051,Z 270.214,A -85,B 0,C 180,E1 -3628.744,E2 -3628.744} C_VEL
LIN {X 0,Y 545.046,Z 270.214,A -85,B 0,C 180,E1 -3631.679,E2 -3631.679} C_VEL
LIN {X 0,Y 545.034,Z 270.217,A -85,B 0,C 180,E1 -3634.566,E2 -3634.566} C_VEL
LIN {X 0,Y 545,Z 270.217,A -85,B 0,C 180,E1 -3637.307,E2 -3637.307} C_VEL
LIN {X 0,Y 545.048,Z 270.215,A -85,B 0,C 180,E1 -3640.144,E2 -3640.144} C_VEL
LIN {X 0,Y 545.014,Z 270.216,A -85,B 0,C 180,E1 -3643.113,E2 -3643.113} C_VEL
LIN {X 0,Y 545.019,Z 270.221,A -85,B 0,C 180,E1 -3646.23,E2 -3646.23} C_VEL
LIN {X 0,Y 545.02,Z 270.215,A -85,B 0,C 180,E1 -3648.881,E2 -3648.881} C_VEL
LIN {X 0,Y 545.039,Z 270.22,A -85,B 0,C 180,E1 -3651.763,E2 -3651.763} C_VEL
LIN {X 0,Y 545.02,Z 270.217,A -85,B 0,C 180,E1 -3654.531,E2 -3654.531} C_VEL
LIN {X 0,Y 545.061,Z 270.213,A -85,B 0,C 180,E1 -3657.212,E2 -3657.212} C_VEL
LIN {X 0,Y 545.058,Z 270.219,A -85,B 0,C 180,E1 -3659.811,E2 -3659.811} C_VEL
LIN {X 0,Y 545.051,Z 270.317,A -85,B 0,C 180,E1 -3662.736,E2 -3662.736} C_VEL
LIN {X 0,Y 547.254,Z 280.03,A -85,B 0,C 180,E1 -3664.111,E2 -3664.111} C_VEL
LIN {X 0,Y 546.932,Z 297.564,A -85,B 0,C 180,E1 -3666.348,E2 -3666.348} C_VEL
LIN {X 0,Y 546.517,Z 316.307,A -85,B 0,C 180,E1 -3668.699,E2 -3668.699} C_VEL
LIN {X 0,Y 546.434,Z 321.591,A -85,B 0,C 180,E1 -3669.356,E2 -3669.356} C_VEL
LIN {X 0,Y 548.488,Z 332.56,A -85,B 0,C 180,E1 -3669.587,E2 -3669.587} C_VEL
LIN {X 0,Y 547.733,Z 487.234,A -85,B 0,C 180,E1 -3671.679,E2 -3671.679} C_VEL
LIN {X 0,Y 547.536,Z 502.904,A -85,B 0,C 180,E1 -3672.038,E2 -3672.038} C_VEL
LIN {X 0,Y 547.253,Z 517.771,A -85,B 0,C 180,E1 -3672.532,E2 -3672.532} C_VEL
LIN {X 0,Y 546.954,Z 530.803,A -85,B 0,C 180,E1 -3673.1,E2 -3673.1} C_VEL
LIN {X 0,Y 546.564,Z 544.679,A -85,B 0,C 180,E1 -3673.856,E2 -3673.856} C_VEL
LIN {X 0,Y 546.285,Z 556.615,A -85,B 0,C 180,E1 -3674.652,E2 -3674.652} C_VEL
LIN {X 0,Y 545.914,Z 569.155,A -85,B 0,C 180,E1 -3675.652,E2 -3675.652} C_VEL
LIN {X 0,Y 545.589,Z 580.969,A -85,B 0,C 180,E1 -3676.783,E2 -3676.783} C_VEL
LIN {X 0,Y 545.315,Z 590.906,A -85,B 0,C 180,E1 -3677.911,E2 -3677.911} C_VEL
LIN {X 0,Y 545.136,Z 600.624,A -85,B 0,C 180,E1 -3679.226,E2 -3679.226} C_VEL
LIN {X 0,Y 544.891,Z 608.727,A -85,B 0,C 180,E1 -3680.535,E2 -3680.535} C_VEL
LIN {X 0,Y 544.818,Z 615.424,A -85,B 0,C 180,E1 -3681.843,E2 -3681.843} C_VEL
LIN {X 0,Y 544.7,Z 622.094,A -85,B 0,C 180,E1 -3683.46,E2 -3683.46} C_VEL
LIN {X 0,Y 544.642,Z 626.387,A -85,B 0,C 180,E1 -3684.818,E2 -3684.818} C_VEL
LIN {X 0,Y 544.644,Z 629.888,A -85,B 0,C 180,E1 -3686.301,E2 -3686.301} C_VEL
LIN {X 0,Y 544.568,Z 632.19,A -85,B 0,C 180,E1 -3687.781,E2 -3687.781} C_VEL
LIN {X 0,Y 544.539,Z 633.348,A -85,B 0,C 180,E1 -3689.261,E2 -3689.261} C_VEL
LIN {X 0,Y 544.539,Z 633.347,A -85,B 0,C 180,E1 -3690.739,E2 -3690.739} C_VEL
LIN {X 0,Y 544.568,Z 632.187,A -85,B 0,C 180,E1 -3692.219,E2 -3692.219} C_VEL
LIN {X 0,Y 544.644,Z 629.884,A -85,B 0,C 180,E1 -3693.699,E2 -3693.699} C_VEL
LIN {X 0,Y 544.642,Z 626.387,A -85,B 0,C 180,E1 -3695.182,E2 -3695.182} C_VEL
LIN {X 0,Y 544.697,Z 621.61,A -85,B 0,C 180,E1 -3696.668,E2 -3696.668} C_VEL
LIN {X 0,Y 544.818,Z 615.422,A -85,B 0,C 180,E1 -3698.157,E2 -3698.157} C_VEL
LIN {X 0,Y 544.904,Z 607.645,A -85,B 0,C 180,E1 -3699.652,E2 -3699.652} C_VEL
LIN {X 0,Y 545.15,Z 599.369,A -85,B 0,C 180,E1 -3700.962,E2 -3700.962} C_VEL
LIN {X 0,Y 545.357,Z 589.394,A -85,B 0,C 180,E1 -3702.276,E2 -3702.276} C_VEL
LIN {X 0,Y 545.639,Z 579.188,A -85,B 0,C 180,E1 -3703.405,E2 -3703.405} C_VEL
LIN {X 0,Y 545.972,Z 567.023,A -85,B 0,C 180,E1 -3704.537,E2 -3704.537} C_VEL
LIN {X 0,Y 546.376,Z 553.388,A -85,B 0,C 180,E1 -3705.581,E2 -3705.581} C_VEL
LIN {X 0,Y 546.748,Z 539.889,A -85,B 0,C 180,E1 -3706.426,E2 -3706.426} C_VEL
LIN {X 0,Y 547.064,Z 525.793,A -85,B 0,C 180,E1 -3707.137,E2 -3707.137} C_VEL
LIN {X 0,Y 547.387,Z 511.264,A -85,B 0,C 180,E1 -3707.705,E2 -3707.705} C_VEL
LIN {X 0,Y 547.646,Z 495.272,A -85,B 0,C 180,E1 -3708.158,E2 -3708.158} C_VEL
LIN {X 0,Y 547.806,Z 479.143,A -85,B 0,C 180,E1 -3708.445,E2 -3708.445} C_VEL
LIN {X 0,Y 548.485,Z 332.653,A -85,B 0,C 180,E1 -3710.412,E2 -3710.412} C_VEL
LIN {X 0,Y 546.426,Z 321.51,A -85,B 0,C 180,E1 -3710.655,E2 -3710.655} C_VEL
LIN {X 0,Y 546.909,Z 298.956,A -85,B 0,C 180,E1 -3713.475,E2 -3713.475} C_VEL
LIN {X 0,Y 547.287,Z 281.614,A -85,B 0,C 180,E1 -3715.683,E2 -3715.683} C_VEL
LIN {X 0,Y 546.617,Z 276.861,A -85,B 0,C 180,E1 -3716.331,E2 -3716.331} C_VEL
LIN {X 0,Y 545.051,Z 270.217,A -85,B 0,C 180,E1 -3717.298,E2 -3717.298} C_VEL
LIN {X 0,Y 545.074,Z 270.216,A -85,B 0,C 180,E1 -3720.246,E2 -3720.246} C_VEL
LIN {X 0,Y 545.072,Z 270.209,A -85,B 0,C 180,E1 -3723.061,E2 -3723.061} C_VEL
LIN {X 0,Y 545.016,Z 270.219,A -85,B 0,C 180,E1 -3725.67,E2 -3725.67} C_VEL
LIN {X 0,Y 545.04,Z 270.221,A -85,B 0,C 180,E1 -3728.237,E2 -3728.237} C_VEL
LIN {X 0,Y 545.02,Z 270.216,A -85,B 0,C 180,E1 -3731.119,E2 -3731.119} C_VEL
LIN {X 0,Y 545.022,Z 270.223,A -85,B 0,C 180,E1 -3734.131,E2 -3734.131} C_VEL
LIN {X 0,Y 545.014,Z 270.216,A -85,B 0,C 180,E1 -3736.887,E2 -3736.887} C_VEL
LIN {X 0,Y 545.048,Z 270.219,A -85,B 0,C 180,E1 -3739.856,E2 -3739.856} C_VEL
LIN {X 0,Y 545.006,Z 270.217,A -85,B 0,C 180,E1 -3742.694,E2 -3742.694} C_VEL
LIN {X 0,Y 545.055,Z 270.216,A -85,B 0,C 180,E1 -3745.609,E2 -3745.609} C_VEL
LIN {X 0,Y 545.046,Z 270.214,A -85,B 0,C 180,E1 -3748.321,E2 -3748.321} C_VEL
LIN {X 0,Y 545.051,Z 270.213,A -85,B 0,C 180,E1 -3751.256,E2 -3751.256} C_VEL
LIN {X 0,Y 545.022,Z 270.22,A -85,B 0,C 180,E1 -3753.997,E2 -3753.997} C_VEL
LIN {X 0,Y 545.059,Z 270.21,A -85,B 0,C 180,E1 -3756.44,E2 -3756.44} C_VEL
LIN {X 0,Y 545.076,Z 270.213,A -85,B 0,C 180,E1 -3759.627,E2 -3759.627} C_VEL
LIN {X 0,Y 545.035,Z 270.211,A -85,B 0,C 180,E1 -3762.748,E2 -3762.748} C_VEL
LIN {X 0,Y 545.055,Z 270.214,A -85,B 0,C 180,E1 -3765.819,E2 -3765.819} C_VEL
LIN {X 0,Y 545.052,Z 270.204,A -85,B 0,C 180,E1 -3768.848,E2 -3768.848} C_VEL
LIN {X 0,Y 545.049,Z 270.215,A -85,B 0,C 180,E1 -3771.846,E2 -3771.846} C_VEL
LIN {X 0,Y 545.113,Z 270.203,A -85,B 0,C 180,E1 -3774.08,E2 -3774.08} C_VEL
LIN {X 0,Y 545.036,Z 270.221,A -85,B 0,C 180,E1 -3775.563,E2 -3775.563} C_VEL
LIN {X 0,Y 545.168,Z 270.199,A -85,B 0,C 180,E1 -3777.784,E2 -3777.784} C_VEL
LIN {X 0,Y 545.166,Z 270.198,A -85,B 0,C 180,E1 -3780,E2 -3780} C_VEL
LIN {X 0,Y 545.146,Z 270.201,A -85,B 0,C 180,E1 -3782.956,E2 -3782.956} C_VEL
LIN {X 0,Y 545.119,Z 270.203,A -85,B 0,C 180,E1 -3785.92,E2 -3785.92} C_VEL
LIN {X 0,Y 545.077,Z 270.208,A -85,B 0,C 180,E1 -3788.154,E2 -3788.154} C_VEL
LIN {X 0,Y 545.119,Z 270.207,A -85,B 0,C 180,E1 -3791.533,E2 -3791.533} C_VEL
LIN {X 0,Y 545.064,Z 270.215,A -85,B 0,C 180,E1 -3794.944,E2 -3794.944} C_VEL
LIN {X 0,Y 545.047,Z 270.211,A -85,B 0,C 180,E1 -3798.027,E2 -3798.027} C_VEL
LIN {X 0,Y 545.077,Z 270.203,A -85,B 0,C 180,E1 -3800.373,E2 -3800.373} C_VEL
LIN {X 0,Y 545.06,Z 270.213,A -85,B 0,C 180,E1 -3803.56,E2 -3803.56} C_VEL
LIN {X 0,Y 545.058,Z 270.208,A -85,B 0,C 180,E1 -3806.002,E2 -3806.002} C_VEL
LIN {X 0,Y 545.063,Z 270.211,A -85,B 0,C 180,E1 -3808.746,E2 -3808.746} C_VEL
LIN {X 0,Y 545.047,Z 270.211,A -85,B 0,C 180,E1 -3811.68,E2 -3811.68} C_VEL
LIN {X 0,Y 545.05,Z 270.215,A -85,B 0,C 180,E1 -3814.565,E2 -3814.565} C_VEL
LIN {X 0,Y 545.055,Z 270.217,A -85,B 0,C 180,E1 -3816.971,E2 -3816.971} C_VEL
LIN {X 0,Y 544.345,Z 270.301,A -85,B 0,C 180,E1 -3817.588,E2 -3817.588} C_VEL
LIN {X 0,Y 541.48,Z 270.66,A -85,B 0,C 180,E1 -3818.589,E2 -3818.589} C_VEL
LIN {X 0,Y 539.093,Z 270.954,A -85,B 0,C 180,E1 -3819.395,E2 -3819.395} C_VEL
LIN {X 0,Y 538.083,Z 271.078,A -85,B 0,C 180,E1 -3820.017,E2 -3820.017} C_VEL
LIN {X 0,Y 538.007,Z 271.089,A -85,B 0,C 180,E1 -3820.227,E2 -3820.227} C_VEL
LIN {X 0,Y 538.019,Z 271.094,A -85,B 0,C 180,E1 -3822.988,E2 -3822.988} C_VEL
LIN {X 0,Y 537.996,Z 271.092,A -85,B 0,C 180,E1 -3826.185,E2 -3826.185} C_VEL
LIN {X 0,Y 538.043,Z 271.087,A -85,B 0,C 180,E1 -3829.254,E2 -3829.254} C_VEL
LIN {X 0,Y 537.986,Z 271.092,A -85,B 0,C 180,E1 -3832.123,E2 -3832.123} C_VEL
LIN {X 0,Y 537.998,Z 271.096,A -85,B 0,C 180,E1 -3834.917,E2 -3834.917} C_VEL
LIN {X 0,Y 538.014,Z 271.089,A -85,B 0,C 180,E1 -3837.618,E2 -3837.618} C_VEL
LIN {X 0,Y 538.01,Z 271.094,A -85,B 0,C 180,E1 -3840.239,E2 -3840.239} C_VEL
LIN {X 0,Y 538.061,Z 271.083,A -85,B 0,C 180,E1 -3842.797,E2 -3842.797} C_VEL
LIN {X 0,Y 538.02,Z 271.136,A -85,B 0,C 180,E1 -3845.678,E2 -3845.678} C_VEL
LIN {X 0,Y 539.69,Z 279.281,A -85,B 0,C 180,E1 -3847.005,E2 -3847.005} C_VEL
LIN {X 0,Y 539.429,Z 293.579,A -85,B 0,C 180,E1 -3849.136,E2 -3849.136} C_VEL
LIN {X 0,Y 541.83,Z 305.313,A -85,B 0,C 180,E1 -3849.397,E2 -3849.397} C_VEL
LIN {X 0,Y 541.022,Z 458.81,A -85,B 0,C 180,E1 -3851.508,E2 -3851.508} C_VEL
LIN {X 0,Y 540.799,Z 474.207,A -85,B 0,C 180,E1 -3851.876,E2 -3851.876} C_VEL
LIN {X 0,Y 540.48,Z 489.452,A -85,B 0,C 180,E1 -3852.403,E2 -3852.403} C_VEL
LIN {X 0,Y 540.141,Z 502.141,A -85,B 0,C 180,E1 -3852.977,E2 -3852.977} C_VEL
LIN {X 0,Y 539.726,Z 515.75,A -85,B 0,C 180,E1 -3853.743,E2 -3853.743} C_VEL
LIN {X 0,Y 539.344,Z 528.7,A -85,B 0,C 180,E1 -3854.637,E2 -3854.637} C_VEL
LIN {X 0,Y 538.943,Z 540.911,A -85,B 0,C 180,E1 -3855.655,E2 -3855.655} C_VEL
LIN {X 0,Y 538.596,Z 552.381,A -85,B 0,C 180,E1 -3856.8,E2 -3856.8} C_VEL
LIN {X 0,Y 538.253,Z 563.185,A -85,B 0,C 180,E1 -3858.089,E2 -3858.089} C_VEL
LIN {X 0,Y 538.028,Z 572.791,A -85,B 0,C 180,E1 -3859.463,E2 -3859.463} C_VEL
LIN {X 0,Y 537.838,Z 580.498,A -85,B 0,C 180,E1 -3860.789,E2 -3860.789} C_VEL
LIN {X 0,Y 537.701,Z 586.896,A -85,B 0,C 180,E1 -3862.112,E2 -3862.112} C_VEL
LIN {X 0,Y 537.603,Z 592.324,A -85,B 0,C 180,E1 -3863.483,E2 -3863.483} C_VEL
LIN {X 0,Y 537.574,Z 596.26,A -85,B 0,C 180,E1 -3864.749,E2 -3864.749} C_VEL
LIN {X 0,Y 537.562,Z 599.796,A -85,B 0,C 180,E1 -3866.252,E2 -3866.252} C_VEL
LIN {X 0,Y 537.488,Z 602.138,A -85,B 0,C 180,E1 -3867.752,E2 -3867.752} C_VEL
LIN {X 0,Y 537.437,Z 603.337,A -85,B 0,C 180,E1 -3869.251,E2 -3869.251} C_VEL
LIN {X 0,Y 537.439,Z 603.357,A -85,B 0,C 180,E1 -3870.749,E2 -3870.749} C_VEL
LIN {X 0,Y 537.488,Z 602.237,A -85,B 0,C 180,E1 -3872.248,E2 -3872.248} C_VEL
LIN {X 0,Y 537.563,Z 599.974,A -85,B 0,C 180,E1 -3873.748,E2 -3873.748} C_VEL
LIN {X 0,Y 537.573,Z 596.514,A -85,B 0,C 180,E1 -3875.251,E2 -3875.251} C_VEL
LIN {X 0,Y 537.619,Z 591.776,A -85,B 0,C 180,E1 -3876.756,E2 -3876.756} C_VEL
LIN {X 0,Y 537.734,Z 585.639,A -85,B 0,C 180,E1 -3878.266,E2 -3878.266} C_VEL
LIN {X 0,Y 537.858,Z 577.914,A -85,B 0,C 180,E1 -3879.78,E2 -3879.78} C_VEL
LIN {X 0,Y 538.081,Z 569.677,A -85,B 0,C 180,E1 -3881.107,E2 -3881.107} C_VEL
LIN {X 0,Y 538.347,Z 559.77,A -85,B 0,C 180,E1 -3882.439,E2 -3882.439} C_VEL
LIN {X 0,Y 538.651,Z 549.668,A -85,B 0,C 180,E1 -3883.583,E2 -3883.583} C_VEL
LIN {X 0,Y 539.009,Z 537.643,A -85,B 0,C 180,E1 -3884.729,E2 -3884.729} C_VEL
LIN {X 0,Y 539.513,Z 524.325,A -85,B 0,C 180,E1 -3885.777,E2 -3885.777} C_VEL
LIN {X 0,Y 539.928,Z 510.91,A -85,B 0,C 180,E1 -3886.64,E2 -3886.64} C_VEL
LIN {X 0,Y 540.301,Z 496.018,A -85,B 0,C 180,E1 -3887.407,E2 -3887.407} C_VEL
LIN {X 0,Y 540.645,Z 481.52,A -85,B 0,C 180,E1 -3887.982,E2 -3887.982} C_VEL
LIN {X 0,Y 540.928,Z 466.036,A -85,B 0,C 180,E1 -3888.429,E2 -3888.429} C_VEL
LIN {X 0,Y 541.1,Z 451.1,A -85,B 0,C 180,E1 -3888.706,E2 -3888.706} C_VEL
LIN {X 0,Y 541.815,Z 304.597,A -85,B 0,C 180,E1 -3890.704,E2 -3890.704} C_VEL
LIN {X 0,Y 539.419,Z 293.36,A -85,B 0,C 180,E1 -3890.98,E2 -3890.98} C_VEL
LIN {X 0,Y 539.754,Z 279.874,A -85,B 0,C 180,E1 -3892.993,E2 -3892.993} C_VEL
LIN {X 0,Y 538.04,Z 271.091,A -85,B 0,C 180,E1 -3894.426,E2 -3894.426} C_VEL
LIN {X 0,Y 538.055,Z 271.092,A -85,B 0,C 180,E1 -3897.351,E2 -3897.351} C_VEL
LIN {X 0,Y 538.024,Z 271.089,A -85,B 0,C 180,E1 -3900.443,E2 -3900.443} C_VEL
LIN {X 0,Y 538.043,Z 271.093,A -85,B 0,C 180,E1 -3903.282,E2 -3903.282} C_VEL
LIN {X 0,Y 538.02,Z 271.091,A -85,B 0,C 180,E1 -3906.001,E2 -3906.001} C_VEL
LIN {X 0,Y 538.009,Z 271.092,A -85,B 0,C 180,E1 -3908.829,E2 -3908.829} C_VEL
LIN {X 0,Y 538.025,Z 271.091,A -85,B 0,C 180,E1 -3911.772,E2 -3911.772} C_VEL
LIN {X 0,Y 537.997,Z 271.093,A -85,B 0,C 180,E1 -3914.862,E2 -3914.862} C_VEL
LIN {X 0,Y 538.012,Z 271.095,A -85,B 0,C 180,E1 -3917.213,E2 -3917.213} C_VEL
LIN {X 0,Y 538.013,Z 271.088,A -85,B 0,C 180,E1 -3920.202,E2 -3920.202} C_VEL
LIN {X 0,Y 538.015,Z 271.091,A -85,B 0,C 180,E1 -3923.066,E2 -3923.066} C_VEL
LIN {X 0,Y 538.002,Z 271.09,A -85,B 0,C 180,E1 -3925.825,E2 -3925.825} C_VEL
LIN {X 0,Y 537.998,Z 271.089,A -85,B 0,C 180,E1 -3928.498,E2 -3928.498} C_VEL
LIN {X 0,Y 538.008,Z 271.094,A -85,B 0,C 180,E1 -3931.097,E2 -3931.097} C_VEL
LIN {X 0,Y 538.025,Z 271.087,A -85,B 0,C 180,E1 -3933.632,E2 -3933.632} C_VEL
LIN {X 0,Y 537.998,Z 271.098,A -85,B 0,C 180,E1 -3936.927,E2 -3936.927} C_VEL
LIN {X 0,Y 538.068,Z 271.081,A -85,B 0,C 180,E1 -3940.147,E2 -3940.147} C_VEL
LIN {X 0,Y 538.002,Z 271.093,A -85,B 0,C 180,E1 -3943.298,E2 -3943.298} C_VEL
LIN {X 0,Y 538.042,Z 271.084,A -85,B 0,C 180,E1 -3945.63,E2 -3945.63} C_VEL
LIN {X 0,Y 538.058,Z 271.089,A -85,B 0,C 180,E1 -3948.701,E2 -3948.701} C_VEL
LIN {X 0,Y 538.043,Z 271.083,A -85,B 0,C 180,E1 -3951.739,E2 -3951.739} C_VEL
LIN {X 0,Y 538.134,Z 271.079,A -85,B 0,C 180,E1 -3954.755,E2 -3954.755} C_VEL
LIN {X 0,Y 538.14,Z 271.072,A -85,B 0,C 180,E1 -3957.755,E2 -3957.755} C_VEL
LIN {X 0,Y 538.169,Z 271.076,A -85,B 0,C 180,E1 -3960.748,E2 -3960.748} C_VEL
LIN {X 0,Y 538.109,Z 271.079,A -85,B 0,C 180,E1 -3962.995,E2 -3962.995} C_VEL
LIN {X 0,Y 538.071,Z 271.081,A -85,B 0,C 180,E1 -3965.998,E2 -3965.998} C_VEL
LIN {X 0,Y 538.022,Z 271.092,A -85,B 0,C 180,E1 -3968.261,E2 -3968.261} C_VEL
LIN {X 0,Y 538.069,Z 271.081,A -85,B 0,C 180,E1 -3971.597,E2 -3971.597} C_VEL
LIN {X 0,Y 538.045,Z 271.088,A -85,B 0,C 180,E1 -3974.857,E2 -3974.857} C_VEL
LIN {X 0,Y 537.991,Z 271.097,A -85,B 0,C 180,E1 -3978.272,E2 -3978.272} C_VEL
LIN {X 0,Y 538.022,Z 271.091,A -85,B 0,C 180,E1 -3980.652,E2 -3980.652} C_VEL
LIN {X 0,Y 537.993,Z 271.094,A -85,B 0,C 180,E1 -3983.878,E2 -3983.878} C_VEL
LIN {X 0,Y 537.967,Z 271.101,A -85,B 0,C 180,E1 -3986.371,E2 -3986.371} C_VEL
LIN {X 0,Y 538.018,Z 271.088,A -85,B 0,C 180,E1 -3988.934,E2 -3988.934} C_VEL
LIN {X 0,Y 537.998,Z 271.094,A -85,B 0,C 180,E1 -3991.887,E2 -3991.887} C_VEL
LIN {X 0,Y 537.984,Z 271.095,A -85,B 0,C 180,E1 -3994.616,E2 -3994.616} C_VEL
LIN {X 0,Y 537.97,Z 271.098,A -85,B 0,C 180,E1 -3997.88,E2 -3997.88} C_VEL
LIN {X 0,Y 537.991,Z 271.087,A -85,B 0,C 180,E1 -4000.781,E2 -4000.781} C_VEL
LIN {X 0,Y 538.002,Z 271.097,A -85,B 0,C 180,E1 -4004.073,E2 -4004.073} C_VEL
LIN {X 0,Y 537.963,Z 271.094,A -85,B 0,C 180,E1 -4007.02,E2 -4007.02} C_VEL
LIN {X 0,Y 537.995,Z 271.091,A -85,B 0,C 180,E1 -4009.259,E2 -4009.259} C_VEL
LIN {X 0,Y 537.979,Z 271.098,A -85,B 0,C 180,E1 -4012.122,E2 -4012.122} C_VEL
LIN {X 0,Y 537.986,Z 271.093,A -85,B 0,C 180,E1 -4014.916,E2 -4014.916} C_VEL
LIN {X 0,Y 538.012,Z 271.096,A -85,B 0,C 180,E1 -4017.618,E2 -4017.618} C_VEL
LIN {X 0,Y 538.009,Z 271.095,A -85,B 0,C 180,E1 -4020.239,E2 -4020.239} C_VEL
LIN {X 0,Y 538.035,Z 271.195,A -85,B 0,C 180,E1 -4022.493,E2 -4022.493} C_VEL
LIN {X 0,Y 540.43,Z 281.704,A -85,B 0,C 180,E1 -4024.004,E2 -4024.004} C_VEL
LIN {X 0,Y 540.075,Z 298.77,A -85,B 0,C 180,E1 -4026.21,E2 -4026.21} C_VEL
LIN {X 0,Y 539.597,Z 317.687,A -85,B 0,C 180,E1 -4028.612,E2 -4028.612} C_VEL
LIN {X 0,Y 539.538,Z 321.394,A -85,B 0,C 180,E1 -4029.08,E2 -4029.08} C_VEL
LIN {X 0,Y 541.832,Z 333.172,A -85,B 0,C 180,E1 -4029.336,E2 -4029.336} C_VEL
LIN {X 0,Y 540.998,Z 487.935,A -85,B 0,C 180,E1 -4031.459,E2 -4031.459} C_VEL
LIN {X 0,Y 540.75,Z 503.44,A -85,B 0,C 180,E1 -4031.825,E2 -4031.825} C_VEL
LIN {X 0,Y 540.418,Z 518.802,A -85,B 0,C 180,E1 -4032.352,E2 -4032.352} C_VEL
LIN {X 0,Y 540.086,Z 532.593,A -85,B 0,C 180,E1 -4032.976,E2 -4032.976} C_VEL
LIN {X 0,Y 539.646,Z 546.108,A -85,B 0,C 180,E1 -4033.74,E2 -4033.74} C_VEL
LIN {X 0,Y 539.309,Z 559.211,A -85,B 0,C 180,E1 -4034.65,E2 -4034.65} C_VEL
LIN {X 0,Y 538.889,Z 571.256,A -85,B 0,C 180,E1 -4035.654,E2 -4035.654} C_VEL
LIN {X 0,Y 538.593,Z 582.75,A -85,B 0,C 180,E1 -4036.8,E2 -4036.8} C_VEL
LIN {X 0,Y 538.282,Z 592.39,A -85,B 0,C 180,E1 -4037.942,E2 -4037.942} C_VEL
LIN {X 0,Y 538.068,Z 601.855,A -85,B 0,C 180,E1 -4039.273,E2 -4039.273} C_VEL
LIN {X 0,Y 537.824,Z 609.736,A -85,B 0,C 180,E1 -4040.599,E2 -4040.599} C_VEL
LIN {X 0,Y 537.699,Z 617.09,A -85,B 0,C 180,E1 -4042.112,E2 -4042.112} C_VEL
LIN {X 0,Y 537.622,Z 622.405,A -85,B 0,C 180,E1 -4043.464,E2 -4043.464} C_VEL
LIN {X 0,Y 537.574,Z 626.386,A -85,B 0,C 180,E1 -4044.749,E2 -4044.749} C_VEL
LIN {X 0,Y 537.561,Z 629.887,A -85,B 0,C 180,E1 -4046.252,E2 -4046.252} C_VEL
LIN {X 0,Y 537.487,Z 632.189,A -85,B 0,C 180,E1 -4047.752,E2 -4047.752} C_VEL
LIN {X 0,Y 537.439,Z 633.348,A -85,B 0,C 180,E1 -4049.251,E2 -4049.251} C_VEL
LIN {X 0,Y 537.439,Z 633.347,A -85,B 0,C 180,E1 -4050.749,E2 -4050.749} C_VEL
LIN {X 0,Y 537.487,Z 632.186,A -85,B 0,C 180,E1 -4052.248,E2 -4052.248} C_VEL
LIN {X 0,Y 537.561,Z 629.883,A -85,B 0,C 180,E1 -4053.748,E2 -4053.748} C_VEL
LIN {X 0,Y 537.574,Z 626.387,A -85,B 0,C 180,E1 -4055.251,E2 -4055.251} C_VEL
LIN {X 0,Y 537.618,Z 621.61,A -85,B 0,C 180,E1 -4056.756,E2 -4056.756} C_VEL
LIN {X 0,Y 537.734,Z 615.421,A -85,B 0,C 180,E1 -4058.266,E2 -4058.266} C_VEL
LIN {X 0,Y 537.859,Z 607.644,A -85,B 0,C 180,E1 -4059.78,E2 -4059.78} C_VEL
LIN {X 0,Y 538.101,Z 599.368,A -85,B 0,C 180,E1 -4061.107,E2 -4061.107} C_VEL
LIN {X 0,Y 538.357,Z 589.394,A -85,B 0,C 180,E1 -4062.439,E2 -4062.439} C_VEL
LIN {X 0,Y 538.662,Z 579.187,A -85,B 0,C 180,E1 -4063.582,E2 -4063.582} C_VEL
LIN {X 0,Y 539.028,Z 566.965,A -85,B 0,C 180,E1 -4064.728,E2 -4064.728} C_VEL
LIN {X 0,Y 539.457,Z 554.716,A -85,B 0,C 180,E1 -4065.682,E2 -4065.682} C_VEL
LIN {X 0,Y 539.836,Z 541.342,A -85,B 0,C 180,E1 -4066.546,E2 -4066.546} C_VEL
LIN {X 0,Y 540.212,Z 526.611,A -85,B 0,C 180,E1 -4067.313,E2 -4067.313} C_VEL
LIN {X 0,Y 540.576,Z 512.37,A -85,B 0,C 180,E1 -4067.887,E2 -4067.887} C_VEL
LIN {X 0,Y 540.843,Z 497.504,A -85,B 0,C 180,E1 -4068.332,E2 -4068.332} C_VEL
LIN {X 0,Y 541.034,Z 482.628,A -85,B 0,C 180,E1 -4068.628,E2 -4068.628} C_VEL
LIN {X 0,Y 541.775,Z 332.74,A -85,B 0,C 180,E1 -4070.672,E2 -4070.672} C_VEL
LIN {X 0,Y 539.521,Z 321.315,A -85,B 0,C 180,E1 -4070.932,E2 -4070.932} C_VEL
LIN {X 0,Y 540.046,Z 300.343,A -85,B 0,C 180,E1 -4073.588,E2 -4073.588} C_VEL
LIN {X 0,Y 540.473,Z 283.299,A -85,B 0,C 180,E1 -4075.785,E2 -4075.785} C_VEL
LIN {X 0,Y 539.692,Z 278.243,A -85,B 0,C 180,E1 -4076.487,E2 -4076.487} C_VEL
LIN {X 0,Y 538.009,Z 271.096,A -85,B 0,C 180,E1 -4077.556,E2 -4077.556} C_VEL
LIN {X 0,Y 538.023,Z 271.092,A -85,B 0,C 180,E1 -4080.443,E2 -4080.443} C_VEL
LIN {X 0,Y 538.041,Z 271.085,A -85,B 0,C 180,E1 -4083.282,E2 -4083.282} C_VEL
LIN {X 0,Y 537.982,Z 271.1,A -85,B 0,C 180,E1 -4086.004,E2 -4086.004} C_VEL
LIN {X 0,Y 538.002,Z 271.091,A -85,B 0,C 180,E1 -4088.83,E2 -4088.83} C_VEL
LIN {X 0,Y 537.982,Z 271.099,A -85,B 0,C 180,E1 -4091.873,E2 -4091.873} C_VEL
LIN {X 0,Y 537.985,Z 271.092,A -85,B 0,C 180,E1 -4094.863,E2 -4094.863} C_VEL
LIN {X 0,Y 537.978,Z 271.093,A -85,B 0,C 180,E1 -4097.21,E2 -4097.21} C_VEL
LIN {X 0,Y 538,Z 271.092,A -85,B 0,C 180,E1 -4100.417,E2 -4100.417} C_VEL
LIN {X 0,Y 537.959,Z 271.095,A -85,B 0,C 180,E1 -4103.062,E2 -4103.062} C_VEL
LIN {X 0,Y 537.998,Z 271.098,A -85,B 0,C 180,E1 -4105.825,E2 -4105.825} C_VEL
LIN {X 0,Y 537.996,Z 271.091,A -85,B 0,C 180,E1 -4108.498,E2 -4108.498} C_VEL
LIN {X 0,Y 538.006,Z 271.089,A -85,B 0,C 180,E1 -4111.097,E2 -4111.097} C_VEL
LIN {X 0,Y 537.967,Z 271.1,A -85,B 0,C 180,E1 -4113.629,E2 -4113.629} C_VEL
LIN {X 0,Y 537.993,Z 271.093,A -85,B 0,C 180,E1 -4116.122,E2 -4116.122} C_VEL
LIN {X 0,Y 538.022,Z 271.091,A -85,B 0,C 180,E1 -4119.348,E2 -4119.348} C_VEL
LIN {X 0,Y 537.991,Z 271.094,A -85,B 0,C 180,E1 -4121.728,E2 -4121.728} C_VEL
LIN {X 0,Y 538.024,Z 271.087,A -85,B 0,C 180,E1 -4124.856,E2 -4124.856} C_VEL
LIN {X 0,Y 538.022,Z 271.081,A -85,B 0,C 180,E1 -4127.936,E2 -4127.936} C_VEL
LIN {X 0,Y 538.011,Z 271.088,A -85,B 0,C 180,E1 -4130.981,E2 -4130.981} C_VEL
LIN {X 0,Y 538.052,Z 271.089,A -85,B 0,C 180,E1 -4133.249,E2 -4133.249} C_VEL
LIN {X 0,Y 538.134,Z 271.071,A -85,B 0,C 180,E1 -4134.755,E2 -4134.755} C_VEL
LIN {X 0,Y 538.141,Z 271.074,A -85,B 0,C 180,E1 -4137.755,E2 -4137.755} C_VEL
LIN {X 0,Y 538.136,Z 271.074,A -85,B 0,C 180,E1 -4140,E2 -4140} C_VEL
LIN {X 0,Y 538.114,Z 271.078,A -85,B 0,C 180,E1 -4142.995,E2 -4142.995} C_VEL
LIN {X 0,Y 538.075,Z 271.08,A -85,B 0,C 180,E1 -4145.998,E2 -4145.998} C_VEL
LIN {X 0,Y 538.042,Z 271.084,A -85,B 0,C 180,E1 -4148.261,E2 -4148.261} C_VEL
LIN {X 0,Y 538.069,Z 271.084,A -85,B 0,C 180,E1 -4151.597,E2 -4151.597} C_VEL
LIN {X 0,Y 538.026,Z 271.093,A -85,B 0,C 180,E1 -4155.144,E2 -4155.144} C_VEL
LIN {X 0,Y 538,Z 271.089,A -85,B 0,C 180,E1 -4158.271,E2 -4158.271} C_VEL
LIN {X 0,Y 538.023,Z 271.083,A -85,B 0,C 180,E1 -4160.652,E2 -4160.652} C_VEL
LIN {X 0,Y 537.994,Z 271.091,A -85,B 0,C 180,E1 -4163.878,E2 -4163.878} C_VEL
LIN {X 0,Y 538.025,Z 271.085,A -85,B 0,C 180,E1 -4166.368,E2 -4166.368} C_VEL
LIN {X 0,Y 538.019,Z 271.091,A -85,B 0,C 180,E1 -4168.934,E2 -4168.934} C_VEL
LIN {X 0,Y 537.999,Z 271.088,A -85,B 0,C 180,E1 -4171.888,E2 -4171.888} C_VEL
LIN {X 0,Y 538,Z 271.094,A -85,B 0,C 180,E1 -4174.618,E2 -4174.618} C_VEL
LIN {X 0,Y 537.994,Z 271.094,A -85,B 0,C 180,E1 -4177.171,E2 -4177.171} C_VEL
LIN {X 0,Y 538.007,Z 271.089,A -85,B 0,C 180,E1 -4180.227,E2 -4180.227} C_VEL
LIN {X 0,Y 537.357,Z 271.178,A -85,B 0,C 180,E1 -4180.853,E2 -4180.853} C_VEL
LIN {X 0,Y 534.508,Z 271.531,A -85,B 0,C 180,E1 -4181.867,E2 -4181.867} C_VEL
LIN {X 0,Y 532.084,Z 271.833,A -85,B 0,C 180,E1 -4182.685,E2 -4182.685} C_VEL
LIN {X 0,Y 531.035,Z 271.96,A -85,B 0,C 180,E1 -4183.316,E2 -4183.316} C_VEL
LIN {X 0,Y 530.945,Z 271.969,A -85,B 0,C 180,E1 -4183.529,E2 -4183.529} C_VEL
LIN {X 0,Y 530.948,Z 271.974,A -85,B 0,C 180,E1 -4186.505,E2 -4186.505} C_VEL
LIN {X 0,Y 530.978,Z 271.971,A -85,B 0,C 180,E1 -4188.977,E2 -4188.977} C_VEL
LIN {X 0,Y 530.95,Z 271.967,A -85,B 0,C 180,E1 -4191.53,E2 -4191.53} C_VEL
LIN {X 0,Y 530.953,Z 271.972,A -85,B 0,C 180,E1 -4194.381,E2 -4194.381} C_VEL
LIN {X 0,Y 530.963,Z 271.97,A -85,B 0,C 180,E1 -4197.134,E2 -4197.134} C_VEL
LIN {X 0,Y 530.966,Z 271.968,A -85,B 0,C 180,E1 -4199.804,E2 -4199.804} C_VEL
LIN {X 0,Y 531.012,Z 271.964,A -85,B 0,C 180,E1 -4202.468,E2 -4202.468} C_VEL
LIN {X 0,Y 531.001,Z 271.988,A -85,B 0,C 180,E1 -4205.439,E2 -4205.439} C_VEL
LIN {X 0,Y 532.813,Z 280.797,A -85,B 0,C 180,E1 -4206.896,E2 -4206.896} C_VEL
LIN {X 0,Y 532.567,Z 293.697,A -85,B 0,C 180,E1 -4208.849,E2 -4208.849} C_VEL
LIN {X 0,Y 535.235,Z 306.506,A -85,B 0,C 180,E1 -4209.145,E2 -4209.145} C_VEL
LIN {X 0,Y 534.298,Z 458.816,A -85,B 0,C 180,E1 -4211.263,E2 -4211.263} C_VEL
LIN {X 0,Y 534.082,Z 473.591,A -85,B 0,C 180,E1 -4211.615,E2 -4211.615} C_VEL
LIN {X 0,Y 533.765,Z 488.458,A -85,B 0,C 180,E1 -4212.125,E2 -4212.125} C_VEL
LIN {X 0,Y 533.338,Z 502.357,A -85,B 0,C 180,E1 -4212.754,E2 -4212.754} C_VEL
LIN {X 0,Y 532.897,Z 515.963,A -85,B 0,C 180,E1 -4213.528,E2 -4213.528} C_VEL
LIN {X 0,Y 532.456,Z 529.537,A -85,B 0,C 180,E1 -4214.481,E2 -4214.481} C_VEL
LIN {X 0,Y 532.039,Z 541.122,A -85,B 0,C 180,E1 -4215.465,E2 -4215.465} C_VEL
LIN {X 0,Y 531.637,Z 552.591,A -85,B 0,C 180,E1 -4216.624,E2 -4216.624} C_VEL
LIN {X 0,Y 531.293,Z 562.242,A -85,B 0,C 180,E1 -4217.781,E2 -4217.781} C_VEL
LIN {X 0,Y 531.05,Z 571.696,A -85,B 0,C 180,E1 -4219.13,E2 -4219.13} C_VEL
LIN {X 0,Y 530.788,Z 580.568,A -85,B 0,C 180,E1 -4220.666,E2 -4220.666} C_VEL
LIN {X 0,Y 530.642,Z 586.917,A -85,B 0,C 180,E1 -4222.006,E2 -4222.006} C_VEL
LIN {X 0,Y 530.522,Z 592.631,A -85,B 0,C 180,E1 -4223.489,E2 -4223.489} C_VEL
LIN {X 0,Y 530.509,Z 596.261,A -85,B 0,C 180,E1 -4224.679,E2 -4224.679} C_VEL
LIN {X 0,Y 530.481,Z 599.796,A -85,B 0,C 180,E1 -4226.202,E2 -4226.202} C_VEL
LIN {X 0,Y 530.409,Z 602.137,A -85,B 0,C 180,E1 -4227.722,E2 -4227.722} C_VEL
LIN {X 0,Y 530.34,Z 603.337,A -85,B 0,C 180,E1 -4229.241,E2 -4229.241} C_VEL
LIN {X 0,Y 530.341,Z 603.357,A -85,B 0,C 180,E1 -4230.759,E2 -4230.759} C_VEL
LIN {X 0,Y 530.409,Z 602.236,A -85,B 0,C 180,E1 -4232.278,E2 -4232.278} C_VEL
LIN {X 0,Y 530.482,Z 599.972,A -85,B 0,C 180,E1 -4233.798,E2 -4233.798} C_VEL
LIN {X 0,Y 530.507,Z 596.512,A -85,B 0,C 180,E1 -4235.321,E2 -4235.321} C_VEL
LIN {X 0,Y 530.55,Z 591.773,A -85,B 0,C 180,E1 -4236.847,E2 -4236.847} C_VEL
LIN {X 0,Y 530.665,Z 585.664,A -85,B 0,C 180,E1 -4238.376,E2 -4238.376} C_VEL
LIN {X 0,Y 530.814,Z 577.998,A -85,B 0,C 180,E1 -4239.911,E2 -4239.911} C_VEL
LIN {X 0,Y 531.06,Z 569.819,A -85,B 0,C 180,E1 -4241.256,E2 -4241.256} C_VEL
LIN {X 0,Y 531.373,Z 559.969,A -85,B 0,C 180,E1 -4242.605,E2 -4242.605} C_VEL
LIN {X 0,Y 531.708,Z 549.867,A -85,B 0,C 180,E1 -4243.763,E2 -4243.763} C_VEL
LIN {X 0,Y 532.115,Z 537.84,A -85,B 0,C 180,E1 -4244.924,E2 -4244.924} C_VEL
LIN {X 0,Y 532.607,Z 525.78,A -85,B 0,C 180,E1 -4245.89,E2 -4245.89} C_VEL
LIN {X 0,Y 533.04,Z 512.679,A -85,B 0,C 180,E1 -4246.763,E2 -4246.763} C_VEL
LIN {X 0,Y 533.402,Z 500.205,A -85,B 0,C 180,E1 -4247.442,E2 -4247.442} C_VEL
LIN {X 0,Y 533.838,Z 485.612,A -85,B 0,C 180,E1 -4248.071,E2 -4248.071} C_VEL
LIN {X 0,Y 534.129,Z 470.18,A -85,B 0,C 180,E1 -4248.565,E2 -4248.565} C_VEL
LIN {X 0,Y 534.321,Z 456.198,A -85,B 0,C 180,E1 -4248.871,E2 -4248.871} C_VEL
LIN {X 0,Y 535.209,Z 306.03,A -85,B 0,C 180,E1 -4250.953,E2 -4250.953} C_VEL
LIN {X 0,Y 532.575,Z 293.599,A -85,B 0,C 180,E1 -4251.255,E2 -4251.255} C_VEL
LIN {X 0,Y 532.893,Z 281.517,A -85,B 0,C 180,E1 -4253.08,E2 -4253.08} C_VEL
LIN {X 0,Y 531.031,Z 271.964,A -85,B 0,C 180,E1 -4254.664,E2 -4254.664} C_VEL
LIN {X 0,Y 531.012,Z 271.968,A -85,B 0,C 180,E1 -4257.595,E2 -4257.595} C_VEL
LIN {X 0,Y 530.972,Z 271.968,A -85,B 0,C 180,E1 -4260.644,E2 -4260.644} C_VEL
LIN {X 0,Y 530.987,Z 271.969,A -85,B 0,C 180,E1 -4263.772,E2 -4263.772} C_VEL
LIN {X 0,Y 530.962,Z 271.969,A -85,B 0,C 180,E1 -4266.557,E2 -4266.557} C_VEL
LIN {X 0,Y 530.974,Z 271.966,A -85,B 0,C 180,E1 -4269.853,E2 -4269.853} C_VEL
LIN {X 0,Y 530.972,Z 271.966,A -85,B 0,C 180,E1 -4272.456,E2 -4272.456} C_VEL
LIN {X 0,Y 530.969,Z 271.97,A -85,B 0,C 180,E1 -4275.621,E2 -4275.621} C_VEL
LIN {X 0,Y 530.985,Z 271.959,A -85,B 0,C 180,E1 -4278.563,E2 -4278.563} C_VEL
LIN {X 0,Y 530.946,Z 271.971,A -85,B 0,C 180,E1 -4281.528,E2 -4281.528} C_VEL
LIN {X 0,Y 530.945,Z 271.966,A -85,B 0,C 180,E1 -4284.379,E2 -4284.379} C_VEL
LIN {X 0,Y 530.957,Z 271.974,A -85,B 0,C 180,E1 -4287.133,E2 -4287.133} C_VEL
LIN {X 0,Y 530.95,Z 271.964,A -85,B 0,C 180,E1 -4289.802,E2 -4289.802} C_VEL
LIN {X 0,Y 531,Z 271.963,A -85,B 0,C 180,E1 -4292.467,E2 -4292.467} C_VEL
LIN {X 0,Y 530.957,Z 271.973,A -85,B 0,C 180,E1 -4294.94,E2 -4294.94} C_VEL
LIN {X 0,Y 530.964,Z 271.964,A -85,B 0,C 180,E1 -4297.898,E2 -4297.898} C_VEL
LIN {X 0,Y 530.971,Z 271.97,A -85,B 0,C 180,E1 -4300.676,E2 -4300.676} C_VEL
LIN {X 0,Y 530.959,Z 271.973,A -85,B 0,C 180,E1 -4303.07,E2 -4303.07} C_VEL
LIN {X 0,Y 531,Z 271.962,A -85,B 0,C 180,E1 -4305.435,E2 -4305.435} C_VEL
LIN {X 0,Y 531.017,Z 271.964,A -85,B 0,C 180,E1 -4308.549,E2 -4308.549} C_VEL
LIN {X 0,Y 531.018,Z 271.958,A -85,B 0,C 180,E1 -4311.629,E2 -4311.629} C_VEL
LIN {X 0,Y 531.092,Z 271.957,A -85,B 0,C 180,E1 -4314.685,E2 -4314.685} C_VEL
LIN {X 0,Y 531.114,Z 271.947,A -85,B 0,C 180,E1 -4317.725,E2 -4317.725} C_VEL
LIN {X 0,Y 531.138,Z 271.952,A -85,B 0,C 180,E1 -4320.758,E2 -4320.758} C_VEL
LIN {X 0,Y 531.075,Z 271.955,A -85,B 0,C 180,E1 -4323.034,E2 -4323.034} C_VEL
LIN {X 0,Y 531.032,Z 271.959,A -85,B 0,C 180,E1 -4326.078,E2 -4326.078} C_VEL
LIN {X 0,Y 530.972,Z 271.972,A -85,B 0,C 180,E1 -4328.372,E2 -4328.372} C_VEL
LIN {X 0,Y 531.033,Z 271.958,A -85,B 0,C 180,E1 -4331.669,E2 -4331.669} C_VEL
LIN {X 0,Y 531.017,Z 271.962,A -85,B 0,C 180,E1 -4334.956,E2 -4334.956} C_VEL
LIN {X 0,Y 530.958,Z 271.967,A -85,B 0,C 180,E1 -4337.724,E2 -4337.724} C_VEL
LIN {X 0,Y 531.011,Z 271.966,A -85,B 0,C 180,E1 -4340.128,E2 -4340.128} C_VEL
LIN {X 0,Y 530.929,Z 271.977,A -85,B 0,C 180,E1 -4342.574,E2 -4342.574} C_VEL
LIN {X 0,Y 530.933,Z 271.97,A -85,B 0,C 180,E1 -4345.061,E2 -4345.061} C_VEL
LIN {X 0,Y 530.949,Z 271.969,A -85,B 0,C 180,E1 -4347.599,E2 -4347.599} C_VEL
LIN {X 0,Y 530.941,Z 271.978,A -85,B 0,C 180,E1 -4350.199,E2 -4350.199} C_VEL
LIN {X 0,Y 530.955,Z 271.966,A -85,B 0,C 180,E1 -4352.867,E2 -4352.867} C_VEL
LIN {X 0,Y 530.918,Z 271.974,A -85,B 0,C 180,E1 -4355.623,E2 -4355.623} C_VEL
LIN {X 0,Y 530.95,Z 271.969,A -85,B 0,C 180,E1 -4358.653,E2 -4358.653} C_VEL
LIN {X 0,Y 530.954,Z 271.964,A -85,B 0,C 180,E1 -4361.439,E2 -4361.439} C_VEL
LIN {X 0,Y 530.957,Z 271.97,A -85,B 0,C 180,E1 -4364.55,E2 -4364.55} C_VEL
LIN {X 0,Y 530.911,Z 271.976,A -85,B 0,C 180,E1 -4367.538,E2 -4367.538} C_VEL
LIN {X 0,Y 530.962,Z 271.968,A -85,B 0,C 180,E1 -4370.556,E2 -4370.556} C_VEL
LIN {X 0,Y 530.93,Z 271.973,A -85,B 0,C 180,E1 -4373.441,E2 -4373.441} C_VEL
LIN {X 0,Y 530.994,Z 271.966,A -85,B 0,C 180,E1 -4376.495,E2 -4376.495} C_VEL
LIN {X 0,Y 530.97,Z 271.968,A -85,B 0,C 180,E1 -4379.356,E2 -4379.356} C_VEL
LIN {X 0,Y 530.969,Z 272.081,A -85,B 0,C 180,E1 -4382.242,E2 -4382.242} C_VEL
LIN {X 0,Y 533.621,Z 283.742,A -85,B 0,C 180,E1 -4383.944,E2 -4383.944} C_VEL
LIN {X 0,Y 533.137,Z 303.303,A -85,B 0,C 180,E1 -4386.5,E2 -4386.5} C_VEL
LIN {X 0,Y 532.635,Z 321.196,A -85,B 0,C 180,E1 -4388.796,E2 -4388.796} C_VEL
LIN {X 0,Y 535.193,Z 334.234,A -85,B 0,C 180,E1 -4389.086,E2 -4389.086} C_VEL
LIN {X 0,Y 534.285,Z 487.637,A -85,B 0,C 180,E1 -4391.215,E2 -4391.215} C_VEL
LIN {X 0,Y 533.994,Z 503.237,A -85,B 0,C 180,E1 -4391.587,E2 -4391.587} C_VEL
LIN {X 0,Y 533.644,Z 518.599,A -85,B 0,C 180,E1 -4392.121,E2 -4392.121} C_VEL
LIN {X 0,Y 533.255,Z 532.388,A -85,B 0,C 180,E1 -4392.751,E2 -4392.751} C_VEL
LIN {X 0,Y 532.776,Z 545.903,A -85,B 0,C 180,E1 -4393.525,E2 -4393.525} C_VEL
LIN {X 0,Y 532.412,Z 558.536,A -85,B 0,C 180,E1 -4394.411,E2 -4394.411} C_VEL
LIN {X 0,Y 531.947,Z 571.051,A -85,B 0,C 180,E1 -4395.462,E2 -4395.462} C_VEL
LIN {X 0,Y 531.58,Z 582.574,A -85,B 0,C 180,E1 -4396.623,E2 -4396.623} C_VEL
LIN {X 0,Y 531.254,Z 592.274,A -85,B 0,C 180,E1 -4397.78,E2 -4397.78} C_VEL
LIN {X 0,Y 531.051,Z 601.804,A -85,B 0,C 180,E1 -4399.13,E2 -4399.13} C_VEL
LIN {X 0,Y 530.764,Z 609.735,A -85,B 0,C 180,E1 -4400.473,E2 -4400.473} C_VEL
LIN {X 0,Y 530.639,Z 617.09,A -85,B 0,C 180,E1 -4402.006,E2 -4402.006} C_VEL
LIN {X 0,Y 530.542,Z 622.707,A -85,B 0,C 180,E1 -4403.469,E2 -4403.469} C_VEL
LIN {X 0,Y 530.508,Z 626.386,A -85,B 0,C 180,E1 -4404.679,E2 -4404.679} C_VEL
LIN {X 0,Y 530.48,Z 629.887,A -85,B 0,C 180,E1 -4406.202,E2 -4406.202} C_VEL
LIN {X 0,Y 530.408,Z 632.189,A -85,B 0,C 180,E1 -4407.722,E2 -4407.722} C_VEL
LIN {X 0,Y 530.341,Z 633.347,A -85,B 0,C 180,E1 -4409.241,E2 -4409.241} C_VEL
LIN {X 0,Y 530.341,Z 633.347,A -85,B 0,C 180,E1 -4410.759,E2 -4410.759} C_VEL
LIN {X 0,Y 530.408,Z 632.185,A -85,B 0,C 180,E1 -4412.278,E2 -4412.278} C_VEL
LIN {X 0,Y 530.48,Z 629.882,A -85,B 0,C 180,E1 -4413.798,E2 -4413.798} C_VEL
LIN {X 0,Y 530.508,Z 626.387,A -85,B 0,C 180,E1 -4415.321,E2 -4415.321} C_VEL
LIN {X 0,Y 530.549,Z 621.61,A -85,B 0,C 180,E1 -4416.847,E2 -4416.847} C_VEL
LIN {X 0,Y 530.665,Z 615.42,A -85,B 0,C 180,E1 -4418.376,E2 -4418.376} C_VEL
LIN {X 0,Y 530.808,Z 607.632,A -85,B 0,C 180,E1 -4419.911,E2 -4419.911} C_VEL
LIN {X 0,Y 531.056,Z 599.299,A -85,B 0,C 180,E1 -4421.256,E2 -4421.256} C_VEL
LIN {X 0,Y 531.347,Z 589.258,A -85,B 0,C 180,E1 -4422.605,E2 -4422.605} C_VEL
LIN {X 0,Y 531.685,Z 578.99,A -85,B 0,C 180,E1 -4423.764,E2 -4423.764} C_VEL
LIN {X 0,Y 532.102,Z 566.76,A -85,B 0,C 180,E1 -4424.925,E2 -4424.925} C_VEL
LIN {X 0,Y 532.558,Z 553.285,A -85,B 0,C 180,E1 -4425.981,E2 -4425.981} C_VEL
LIN {X 0,Y 533.056,Z 539.511,A -85,B 0,C 180,E1 -4426.861,E2 -4426.861} C_VEL
LIN {X 0,Y 533.431,Z 525.385,A -85,B 0,C 180,E1 -4427.589,E2 -4427.589} C_VEL
LIN {X 0,Y 533.818,Z 510.856,A -85,B 0,C 180,E1 -4428.171,E2 -4428.171} C_VEL
LIN {X 0,Y 534.126,Z 495.323,A -85,B 0,C 180,E1 -4428.623,E2 -4428.623} C_VEL
LIN {X 0,Y 534.363,Z 478.966,A -85,B 0,C 180,E1 -4428.923,E2 -4428.923} C_VEL
LIN {X 0,Y 535.134,Z 333.795,A -85,B 0,C 180,E1 -4430.923,E2 -4430.923} C_VEL
LIN {X 0,Y 532.632,Z 321.133,A -85,B 0,C 180,E1 -4431.212,E2 -4431.212} C_VEL
LIN {X 0,Y 533.246,Z 300.156,A -85,B 0,C 180,E1 -4433.908,E2 -4433.908} C_VEL
LIN {X 0,Y 533.608,Z 283.766,A -85,B 0,C 180,E1 -4436.054,E2 -4436.054} C_VEL
LIN {X 0,Y 530.95,Z 271.976,A -85,B 0,C 180,E1 -4437.786,E2 -4437.786} C_VEL
LIN {X 0,Y 530.97,Z 271.969,A -85,B 0,C 180,E1 -4440.644,E2 -4440.644} C_VEL
LIN {X 0,Y 530.981,Z 271.969,A -85,B 0,C 180,E1 -4443.772,E2 -4443.772} C_VEL
LIN {X 0,Y 530.93,Z 271.974,A -85,B 0,C 180,E1 -4446.559,E2 -4446.559} C_VEL
LIN {X 0,Y 530.962,Z 271.969,A -85,B 0,C 180,E1 -4449.444,E2 -4449.444} C_VEL
LIN {X 0,Y 530.911,Z 271.977,A -85,B 0,C 180,E1 -4452.462,E2 -4452.462} C_VEL
LIN {X 0,Y 530.957,Z 271.97,A -85,B 0,C 180,E1 -4455.45,E2 -4455.45} C_VEL
LIN {X 0,Y 530.954,Z 271.969,A -85,B 0,C 180,E1 -4458.561,E2 -4458.561} C_VEL
LIN {X 0,Y 530.94,Z 271.973,A -85,B 0,C 180,E1 -4461.528,E2 -4461.528} C_VEL
LIN {X 0,Y 530.921,Z 271.973,A -85,B 0,C 180,E1 -4464.377,E2 -4464.377} C_VEL
LIN {X 0,Y 530.955,Z 271.967,A -85,B 0,C 180,E1 -4467.133,E2 -4467.133} C_VEL
LIN {X 0,Y 530.941,Z 271.976,A -85,B 0,C 180,E1 -4469.801,E2 -4469.801} C_VEL
LIN {X 0,Y 530.95,Z 271.967,A -85,B 0,C 180,E1 -4472.478,E2 -4472.478} C_VEL
LIN {X 0,Y 530.933,Z 271.97,A -85,B 0,C 180,E1 -4474.939,E2 -4474.939} C_VEL
LIN {X 0,Y 530.964,Z 271.971,A -85,B 0,C 180,E1 -4477.898,E2 -4477.898} C_VEL
LIN {X 0,Y 530.965,Z 271.96,A -85,B 0,C 180,E1 -4480.676,E2 -4480.676} C_VEL
LIN {X 0,Y 530.939,Z 271.968,A -85,B 0,C 180,E1 -4483.07,E2 -4483.07} C_VEL
LIN {X 0,Y 530.987,Z 271.97,A -85,B 0,C 180,E1 -4485.435,E2 -4485.435} C_VEL
LIN {X 0,Y 530.968,Z 271.956,A -85,B 0,C 180,E1 -4488.548,E2 -4488.548} C_VEL
LIN {X 0,Y 530.967,Z 271.973,A -85,B 0,C 180,E1 -4491.628,E2 -4491.628} C_VEL
LIN {X 0,Y 531.031,Z 271.958,A -85,B 0,C 180,E1 -4493.922,E2 -4493.922} C_VEL
LIN {X 0,Y 530.969,Z 271.973,A -85,B 0,C 180,E1 -4495.445,E2 -4495.445} C_VEL
LIN {X 0,Y 531.114,Z 271.95,A -85,B 0,C 180,E1 -4497.725,E2 -4497.725} C_VEL
LIN {X 0,Y 531.106,Z 271.95,A -85,B 0,C 180,E1 -4500,E2 -4500} C_VEL
LIN {X 0,Y 531.081,Z 271.954,A -85,B 0,C 180,E1 -4503.034,E2 -4503.034} C_VEL
LIN {X 0,Y 531.035,Z 271.956,A -85,B 0,C 180,E1 -4506.078,E2 -4506.078} C_VEL
LIN {X 0,Y 530.994,Z 271.97,A -85,B 0,C 180,E1 -4509.139,E2 -4509.139} C_VEL
LIN {X 0,Y 531.01,Z 271.96,A -85,B 0,C 180,E1 -4512.226,E2 -4512.226} C_VEL
LIN {X 0,Y 530.977,Z 271.971,A -85,B 0,C 180,E1 -4515.35,E2 -4515.35} C_VEL
LIN {X 0,Y 530.961,Z 271.967,A -85,B 0,C 180,E1 -4518.522,E2 -4518.522} C_VEL
LIN {X 0,Y 530.985,Z 271.962,A -85,B 0,C 180,E1 -4520.939,E2 -4520.939} C_VEL
LIN {X 0,Y 530.943,Z 271.969,A -85,B 0,C 180,E1 -4524.226,E2 -4524.226} C_VEL
LIN {X 0,Y 530.986,Z 271.966,A -85,B 0,C 180,E1 -4526.745,E2 -4526.745} C_VEL
LIN {X 0,Y 530.969,Z 271.97,A -85,B 0,C 180,E1 -4529.323,E2 -4529.323} C_VEL
LIN {X 0,Y 530.954,Z 271.966,A -85,B 0,C 180,E1 -4532.101,E2 -4532.101} C_VEL
LIN {X 0,Y 530.959,Z 271.974,A -85,B 0,C 180,E1 -4534.852,E2 -4534.852} C_VEL
LIN {X 0,Y 530.956,Z 271.967,A -85,B 0,C 180,E1 -4537.509,E2 -4537.509} C_VEL
LIN {X 0,Y 530.972,Z 271.967,A -85,B 0,C 180,E1 -4540.434,E2 -4540.434} C_VEL
LIN {X 0,Y 530.953,Z 271.97,A -85,B 0,C 180,E1 -4543.282,E2 -4543.282} C_VEL
LIN {X 0,Y 530.945,Z 271.969,A -85,B 0,C 180,E1 -4543.529,E2 -4543.529} C_VEL
LIN {X 0,Y 530.27,Z 272.054,A -85,B 0,C 180,E1 -4544.163,E2 -4544.163} C_VEL
LIN {X 0,Y 527.426,Z 272.416,A -85,B 0,C 180,E1 -4545.192,E2 -4545.192} C_VEL
LIN {X 0,Y 525.026,Z 272.719,A -85,B 0,C 180,E1 -4546.02,E2 -4546.02} C_VEL
LIN {X 0,Y 523.995,Z 272.844,A -85,B 0,C 180,E1 -4546.66,E2 -4546.66} C_VEL
LIN {X 0,Y 523.909,Z 272.852,A -85,B 0,C 180,E1 -4546.876,E2 -4546.876} C_VEL
LIN {X 0,Y 523.944,Z 272.842,A -85,B 0,C 180,E1 -4549.921,E2 -4549.921} C_VEL
LIN {X 0,Y 523.903,Z 272.852,A -85,B 0,C 180,E1 -4552.869,E2 -4552.869} C_VEL
LIN {X 0,Y 523.919,Z 272.845,A -85,B 0,C 180,E1 -4555.71,E2 -4555.71} C_VEL
LIN {X 0,Y 523.918,Z 272.852,A -85,B 0,C 180,E1 -4558.457,E2 -4558.457} C_VEL
LIN {X 0,Y 523.928,Z 272.847,A -85,B 0,C 180,E1 -4561.126,E2 -4561.126} C_VEL
LIN {X 0,Y 523.983,Z 272.839,A -85,B 0,C 180,E1 -4563.981,E2 -4563.981} C_VEL
LIN {X 0,Y 523.996,Z 273.009,A -85,B 0,C 180,E1 -4565.221,E2 -4565.221} C_VEL
LIN {X 0,Y 525.928,Z 282.319,A -85,B 0,C 180,E1 -4566.784,E2 -4566.784} C_VEL
LIN {X 0,Y 525.763,Z 294.15,A -85,B 0,C 180,E1 -4568.568,E2 -4568.568} C_VEL
LIN {X 0,Y 528.525,Z 306.432,A -85,B 0,C 180,E1 -4568.863,E2 -4568.863} C_VEL
LIN {X 0,Y 527.81,Z 429.194,A -85,B 0,C 180,E1 -4570.58,E2 -4570.58} C_VEL
LIN {X 0,Y 527.579,Z 459.854,A -85,B 0,C 180,E1 -4571.032,E2 -4571.032} C_VEL
LIN {X 0,Y 527.338,Z 474.653,A -85,B 0,C 180,E1 -4571.397,E2 -4571.397} C_VEL
LIN {X 0,Y 526.989,Z 489.886,A -85,B 0,C 180,E1 -4571.937,E2 -4571.937} C_VEL
LIN {X 0,Y 526.555,Z 502.573,A -85,B 0,C 180,E1 -4572.524,E2 -4572.524} C_VEL
LIN {X 0,Y 526.07,Z 516.177,A -85,B 0,C 180,E1 -4573.308,E2 -4573.308} C_VEL
LIN {X 0,Y 525.619,Z 528.882,A -85,B 0,C 180,E1 -4574.207,E2 -4574.207} C_VEL
LIN {X 0,Y 525.131,Z 541.332,A -85,B 0,C 180,E1 -4575.269,E2 -4575.269} C_VEL
LIN {X 0,Y 524.701,Z 552.801,A -85,B 0,C 180,E1 -4576.444,E2 -4576.444} C_VEL
LIN {X 0,Y 524.313,Z 562.451,A -85,B 0,C 180,E1 -4577.616,E2 -4577.616} C_VEL
LIN {X 0,Y 524.035,Z 571.904,A -85,B 0,C 180,E1 -4578.983,E2 -4578.983} C_VEL
LIN {X 0,Y 523.75,Z 580.775,A -85,B 0,C 180,E1 -4580.539,E2 -4580.539} C_VEL
LIN {X 0,Y 523.594,Z 587.123,A -85,B 0,C 180,E1 -4581.898,E2 -4581.898} C_VEL
LIN {X 0,Y 523.46,Z 593.053,A -85,B 0,C 180,E1 -4583.478,E2 -4583.478} C_VEL
LIN {X 0,Y 523.441,Z 596.406,A -85,B 0,C 180,E1 -4584.607,E2 -4584.607} C_VEL
LIN {X 0,Y 523.402,Z 599.908,A -85,B 0,C 180,E1 -4586.151,E2 -4586.151} C_VEL
LIN {X 0,Y 523.332,Z 602.229,A -85,B 0,C 180,E1 -4587.691,E2 -4587.691} C_VEL
LIN {X 0,Y 523.246,Z 603.42,A -85,B 0,C 180,E1 -4589.23,E2 -4589.23} C_VEL
LIN {X 0,Y 523.247,Z 603.439,A -85,B 0,C 180,E1 -4590.77,E2 -4590.77} C_VEL
LIN {X 0,Y 523.333,Z 602.326,A -85,B 0,C 180,E1 -4592.309,E2 -4592.309} C_VEL
LIN {X 0,Y 523.403,Z 600.081,A -85,B 0,C 180,E1 -4593.849,E2 -4593.849} C_VEL
LIN {X 0,Y 523.439,Z 596.65,A -85,B 0,C 180,E1 -4595.393,E2 -4595.393} C_VEL
LIN {X 0,Y 523.482,Z 591.953,A -85,B 0,C 180,E1 -4596.94,E2 -4596.94} C_VEL
LIN {X 0,Y 523.612,Z 585.865,A -85,B 0,C 180,E1 -4598.49,E2 -4598.49} C_VEL
LIN {X 0,Y 523.785,Z 578.198,A -85,B 0,C 180,E1 -4600.045,E2 -4600.045} C_VEL
LIN {X 0,Y 524.054,Z 570.019,A -85,B 0,C 180,E1 -4601.409,E2 -4601.409} C_VEL
LIN {X 0,Y 524.401,Z 560.169,A -85,B 0,C 180,E1 -4602.775,E2 -4602.775} C_VEL
LIN {X 0,Y 524.788,Z 550.065,A -85,B 0,C 180,E1 -4603.949,E2 -4603.949} C_VEL
LIN {X 0,Y 525.234,Z 538.037,A -85,B 0,C 180,E1 -4605.124,E2 -4605.124} C_VEL
LIN {X 0,Y 525.793,Z 524.819,A -85,B 0,C 180,E1 -4606.192,E2 -4606.192} C_VEL
LIN {X 0,Y 526.345,Z 511.295,A -85,B 0,C 180,E1 -4607.082,E2 -4607.082} C_VEL
LIN {X 0,Y 526.759,Z 496.397,A -85,B 0,C 180,E1 -4607.87,E2 -4607.87} C_VEL
LIN {X 0,Y 527.171,Z 481.89,A -85,B 0,C 180,E1 -4608.458,E2 -4608.458} C_VEL
LIN {X 0,Y 527.497,Z 466.065,A -85,B 0,C 180,E1 -4608.923,E2 -4608.923} C_VEL
LIN {X 0,Y 527.689,Z 450.772,A -85,B 0,C 180,E1 -4609.21,E2 -4609.21} C_VEL
LIN {X 0,Y 528.527,Z 306.584,A -85,B 0,C 180,E1 -4611.225,E2 -4611.225} C_VEL
LIN {X 0,Y 525.727,Z 293.867,A -85,B 0,C 180,E1 -4611.535,E2 -4611.535} C_VEL
LIN {X 0,Y 526.007,Z 282.896,A -85,B 0,C 180,E1 -4613.212,E2 -4613.212} C_VEL
LIN {X 0,Y 523.978,Z 272.844,A -85,B 0,C 180,E1 -4614.912,E2 -4614.912} C_VEL
LIN {X 0,Y 523.958,Z 272.844,A -85,B 0,C 180,E1 -4617.999,E2 -4617.999} C_VEL
LIN {X 0,Y 523.942,Z 272.845,A -85,B 0,C 180,E1 -4620.854,E2 -4620.854} C_VEL
LIN {X 0,Y 523.958,Z 272.845,A -85,B 0,C 180,E1 -4623.734,E2 -4623.734} C_VEL
LIN {X 0,Y 523.916,Z 272.847,A -85,B 0,C 180,E1 -4626.403,E2 -4626.403} C_VEL
LIN {X 0,Y 523.916,Z 272.851,A -85,B 0,C 180,E1 -4629.084,E2 -4629.084} C_VEL
LIN {X 0,Y 523.945,Z 272.842,A -85,B 0,C 180,E1 -4632.118,E2 -4632.118} C_VEL
LIN {X 0,Y 523.935,Z 272.85,A -85,B 0,C 180,E1 -4635.309,E2 -4635.309} C_VEL
LIN {X 0,Y 523.948,Z 272.837,A -85,B 0,C 180,E1 -4638.689,E2 -4638.689} C_VEL
LIN {X 0,Y 523.908,Z 272.853,A -85,B 0,C 180,E1 -4641.08,E2 -4641.08} C_VEL
LIN {X 0,Y 523.891,Z 272.845,A -85,B 0,C 180,E1 -4643.824,E2 -4643.824} C_VEL
LIN {X 0,Y 523.904,Z 272.848,A -85,B 0,C 180,E1 -4646.633,E2 -4646.633} C_VEL
LIN {X 0,Y 523.939,Z 272.841,A -85,B 0,C 180,E1 -4649.354,E2 -4649.354} C_VEL
LIN {X 0,Y 523.963,Z 272.838,A -85,B 0,C 180,E1 -4652.281,E2 -4652.281} C_VEL
LIN {X 0,Y 523.9,Z 272.849,A -85,B 0,C 180,E1 -4655.427,E2 -4655.427} C_VEL
LIN {X 0,Y 523.925,Z 272.841,A -85,B 0,C 180,E1 -4657.939,E2 -4657.939} C_VEL
LIN {X 0,Y 523.956,Z 272.841,A -85,B 0,C 180,E1 -4660.407,E2 -4660.407} C_VEL
LIN {X 0,Y 523.935,Z 272.847,A -85,B 0,C 180,E1 -4662.836,E2 -4662.836} C_VEL
LIN {X 0,Y 523.96,Z 272.841,A -85,B 0,C 180,E1 -4665.235,E2 -4665.235} C_VEL
LIN {X 0,Y 524,Z 272.836,A -85,B 0,C 180,E1 -4668.394,E2 -4668.394} C_VEL
LIN {X 0,Y 523.97,Z 272.836,A -85,B 0,C 180,E1 -4671.515,E2 -4671.515} C_VEL
LIN {X 0,Y 524.002,Z 272.833,A -85,B 0,C 180,E1 -4673.84,E2 -4673.84} C_VEL
LIN {X 0,Y 524.024,Z 272.836,A -85,B 0,C 180,E1 -4676.925,E2 -4676.925} C_VEL
LIN {X 0,Y 524.091,Z 272.821,A -85,B 0,C 180,E1 -4680,E2 -4680} C_VEL
LIN {X 0,Y 524.015,Z 272.834,A -85,B 0,C 180,E1 -4683.075,E2 -4683.075} C_VEL
LIN {X 0,Y 523.998,Z 272.836,A -85,B 0,C 180,E1 -4686.159,E2 -4686.159} C_VEL
LIN {X 0,Y 523.936,Z 272.848,A -85,B 0,C 180,E1 -4688.485,E2 -4688.485} C_VEL
LIN {X 0,Y 523.982,Z 272.837,A -85,B 0,C 180,E1 -4691.736,E2 -4691.736} C_VEL
LIN {X 0,Y 523.98,Z 272.838,A -85,B 0,C 180,E1 -4695.052,E2 -4695.052} C_VEL
LIN {X 0,Y 523.901,Z 272.848,A -85,B 0,C 180,E1 -4697.971,E2 -4697.971} C_VEL
LIN {X 0,Y 523.958,Z 272.847,A -85,B 0,C 180,E1 -4700.41,E2 -4700.41} C_VEL
LIN {X 0,Y 523.895,Z 272.849,A -85,B 0,C 180,E1 -4702.894,E2 -4702.894} C_VEL
LIN {X 0,Y 523.883,Z 272.848,A -85,B 0,C 180,E1 -4705.422,E2 -4705.422} C_VEL
LIN {X 0,Y 523.901,Z 272.851,A -85,B 0,C 180,E1 -4708.003,E2 -4708.003} C_VEL
LIN {X 0,Y 523.923,Z 272.845,A -85,B 0,C 180,E1 -4710.853,E2 -4710.853} C_VEL
LIN {X 0,Y 523.915,Z 272.845,A -85,B 0,C 180,E1 -4713.729,E2 -4713.729} C_VEL
LIN {X 0,Y 523.85,Z 272.857,A -85,B 0,C 180,E1 -4716.395,E2 -4716.395} C_VEL
LIN {X 0,Y 523.9,Z 272.845,A -85,B 0,C 180,E1 -4719.086,E2 -4719.086} C_VEL
LIN {X 0,Y 523.901,Z 272.852,A -85,B 0,C 180,E1 -4722.124,E2 -4722.124} C_VEL
LIN {X 0,Y 523.926,Z 272.844,A -85,B 0,C 180,E1 -4725.312,E2 -4725.312} C_VEL
LIN {X 0,Y 523.912,Z 272.846,A -85,B 0,C 180,E1 -4728.695,E2 -4728.695} C_VEL
LIN {X 0,Y 523.897,Z 272.853,A -85,B 0,C 180,E1 -4731.898,E2 -4731.898} C_VEL
LIN {X 0,Y 523.916,Z 272.846,A -85,B 0,C 180,E1 -4734.912,E2 -4734.912} C_VEL
LIN {X 0,Y 523.93,Z 272.85,A -85,B 0,C 180,E1 -4737.681,E2 -4737.681} C_VEL
LIN {X 0,Y 523.949,Z 272.845,A -85,B 0,C 180,E1 -4740.678,E2 -4740.678} C_VEL
LIN {X 0,Y 523.957,Z 272.877,A -85,B 0,C 180,E1 -4741.974,E2 -4741.974} C_VEL
LIN {X 0,Y 526.801,Z 285.777,A -85,B 0,C 180,E1 -4743.881,E2 -4743.881} C_VEL
LIN {X 0,Y 526.205,Z 306.419,A -85,B 0,C 180,E1 -4746.609,E2 -4746.609} C_VEL
LIN {X 0,Y 525.787,Z 321.272,A -85,B 0,C 180,E1 -4748.512,E2 -4748.512} C_VEL
LIN {X 0,Y 528.544,Z 335.975,A -85,B 0,C 180,E1 -4748.838,E2 -4748.838} C_VEL
LIN {X 0,Y 527.569,Z 487.524,A -85,B 0,C 180,E1 -4750.969,E2 -4750.969} C_VEL
LIN {X 0,Y 527.25,Z 503.033,A -85,B 0,C 180,E1 -4751.343,E2 -4751.343} C_VEL
LIN {X 0,Y 526.861,Z 518.395,A -85,B 0,C 180,E1 -4751.883,E2 -4751.883} C_VEL
LIN {X 0,Y 526.436,Z 532.184,A -85,B 0,C 180,E1 -4752.52,E2 -4752.52} C_VEL
LIN {X 0,Y 525.94,Z 545.699,A -85,B 0,C 180,E1 -4753.304,E2 -4753.304} C_VEL
LIN {X 0,Y 525.501,Z 559.078,A -85,B 0,C 180,E1 -4754.258,E2 -4754.258} C_VEL
LIN {X 0,Y 524.953,Z 571.92,A -85,B 0,C 180,E1 -4755.363,E2 -4755.363} C_VEL
LIN {X 0,Y 524.552,Z 584.141,A -85,B 0,C 180,E1 -4756.638,E2 -4756.638} C_VEL
LIN {X 0,Y 524.136,Z 595.01,A -85,B 0,C 180,E1 -4758.005,E2 -4758.005} C_VEL
LIN {X 0,Y 523.926,Z 604.061,A -85,B 0,C 180,E1 -4759.372,E2 -4759.372} C_VEL
LIN {X 0,Y 523.699,Z 611.568,A -85,B 0,C 180,E1 -4760.733,E2 -4760.733} C_VEL
